	LOCAL CONST Robtarget Tr_meulage_motif_2_P33 :=[[45.7417890625,-26.569017578125,5.9224365234375],[-3.19370360057134E-06,0.00176428802739274,-0.00181018821640207,-0.999996805242986],[0,0,0,0],[8.999999E+09,8.999999E+09,8.999999E+09,8.999999E+09,8.999999E+09,8.999999E+09]];
	LOCAL CONST Robtarget Tr_meulage_motif_2_P34 :=[[46.73433984375,-26.69078125,5.9262734375],[-3.19370360057134E-06,0.00176428802739274,-0.00181018821640207,-0.999996805242986],[0,0,0,0],[8.999999E+09,8.999999E+09,8.999999E+09,8.999999E+09,8.999999E+09,8.999999E+09]];
	LOCAL CONST Robtarget Tr_meulage_motif_2_P35 :=[[47.72689453125,-26.81254296875,5.93011083984375],[-3.19370360057134E-06,0.00176428802739274,-0.00181018821640207,-0.999996805242986],[0,0,0,0],[8.999999E+09,8.999999E+09,8.999999E+09,8.999999E+09,8.999999E+09,8.999999E+09]];
	LOCAL CONST Robtarget Tr_meulage_motif_2_P36 :=[[48.72553515625,-26.823689453125,5.9303427734375],[-3.19370360057134E-06,0.00176428802739274,-0.00181018821640207,-0.999996805242986],[0,0,0,0],[8.999999E+09,8.999999E+09,8.999999E+09,8.999999E+09,8.999999E+09,8.999999E+09]];
	LOCAL CONST Robtarget Tr_meulage_motif_2_P37 :=[[49.69071484375,-26.72943359375,5.92714501953125],[-3.19370360057134E-06,0.00176428802739274,-0.00181018821640207,-0.999996805242986],[0,0,0,0],[8.999999E+09,8.999999E+09,8.999999E+09,8.999999E+09,8.999999E+09,8.999999E+09]];
	LOCAL CONST Robtarget Tr_meulage_motif_2_P38 :=[[50.57019921875,-26.563587890625,5.92162548828125],[-3.19370360057134E-06,0.00176428802739274,-0.00181018821640207,-0.999996805242986],[0,0,0,0],[8.999999E+09,8.999999E+09,8.999999E+09,8.999999E+09,8.999999E+09,8.999999E+09]];
	LOCAL CONST Robtarget Tr_meulage_motif_2_P39 :=[[51.3481640625,-26.3811640625,5.9155791015625],[-3.19370360057134E-06,0.00176428802739274,-0.00181018821640207,-0.999996805242986],[0,0,0,0],[8.999999E+09,8.999999E+09,8.999999E+09,8.999999E+09,8.999999E+09,8.999999E+09]];
	LOCAL CONST Robtarget Tr_meulage_motif_2_P40 :=[[52.5160859375,-25.904021484375,5.89987841796875],[-3.19370360057134E-06,0.00176428802739274,-0.00181018821640207,-0.999996805242986],[0,0,0,0],[8.999999E+09,8.999999E+09,8.999999E+09,8.999999E+09,8.999999E+09,8.999999E+09]];
	LOCAL CONST Robtarget Tr_meulage_motif_2_P41 :=[[53.63559765625,-25.187794921875,5.87639306640625],[-3.19370360057134E-06,0.00176428802739274,-0.00181018821640207,-0.999996805242986],[0,0,0,0],[8.999999E+09,8.999999E+09,8.999999E+09,8.999999E+09,8.999999E+09,8.999999E+09]];
	LOCAL CONST Robtarget Tr_meulage_motif_2_P42 :=[[54.601671875,-24.275298828125,5.84653271484375],[-3.19370360057134E-06,0.00176428802739274,-0.00181018821640207,-0.999996805242986],[0,0,0,0],[8.999999E+09,8.999999E+09,8.999999E+09,8.999999E+09,8.999999E+09,8.999999E+09]];
	LOCAL CONST Robtarget Tr_meulage_motif_2_P43 :=[[55.22216796875,-23.227451171875,5.8123076171875],[-3.19370360057134E-06,0.00176428802739274,-0.00181018821640207,-0.999996805242986],[0,0,0,0],[8.999999E+09,8.999999E+09,8.999999E+09,8.999999E+09,8.999999E+09,8.999999E+09]];
	LOCAL CONST Robtarget Tr_meulage_motif_2_P44 :=[[55.33381640625,-22.540328125,5.7899033203125],[-3.19370360057134E-06,0.00176428802739274,-0.00181018821640207,-0.999996805242986],[0,0,0,0],[8.999999E+09,8.999999E+09,8.999999E+09,8.999999E+09,8.999999E+09,8.999999E+09]];
	LOCAL CONST Robtarget Tr_meulage_motif_2_P45 :=[[55.41437109375,-21.8843515625,5.768517578125],[-3.19370360057134E-06,0.00176428802739274,-0.00181018821640207,-0.999996805242986],[0,0,0,0],[8.999999E+09,8.999999E+09,8.999999E+09,8.999999E+09,8.999999E+09,8.999999E+09]];
	LOCAL CONST Robtarget Tr_meulage_motif_2_P46 :=[[55.44044140625,-21.221849609375,5.7469267578125],[-3.19370360057134E-06,0.00176428802739274,-0.00181018821640207,-0.999996805242986],[0,0,0,0],[8.999999E+09,8.999999E+09,8.999999E+09,8.999999E+09,8.999999E+09,8.999999E+09]];
	LOCAL CONST Robtarget Tr_meulage_motif_2_P47 :=[[55.08015234375,-20.068220703125,5.70938330078125],[-3.19370360057134E-06,0.00176428802739274,-0.00181018821640207,-0.999996805242986],[0,0,0,0],[8.999999E+09,8.999999E+09,8.999999E+09,8.999999E+09,8.999999E+09,8.999999E+09]];
	LOCAL CONST Robtarget Tr_meulage_motif_2_P48 :=[[54.35253515625,-18.9653203125,5.673541015625],[-3.19370360057134E-06,0.00176428802739274,-0.00181018821640207,-0.999996805242986],[0,0,0,0],[8.999999E+09,8.999999E+09,8.999999E+09,8.999999E+09,8.999999E+09,8.999999E+09]];
	LOCAL CONST Robtarget Tr_meulage_motif_2_P49 :=[[53.43773046875,-18.018443359375,5.64280712890625],[-3.19370360057134E-06,0.00176428802739274,-0.00181018821640207,-0.999996805242986],[0,0,0,0],[8.999999E+09,8.999999E+09,8.999999E+09,8.999999E+09,8.999999E+09,8.999999E+09]];
	LOCAL CONST Robtarget Tr_meulage_motif_2_P50 :=[[52.80396484375,-17.542185546875,5.62737158203125],[-3.19370360057134E-06,0.00176428802739274,-0.00181018821640207,-0.999996805242986],[0,0,0,0],[8.999999E+09,8.999999E+09,8.999999E+09,8.999999E+09,8.999999E+09,8.999999E+09]];
	LOCAL CONST Robtarget Tr_meulage_motif_2_P51 :=[[51.713828125,-16.9175234375,5.60716015625],[-3.19370360057134E-06,0.00176428802739274,-0.00181018821640207,-0.999996805242986],[0,0,0,0],[8.999999E+09,8.999999E+09,8.999999E+09,8.999999E+09,8.999999E+09,8.999999E+09]];
	LOCAL CONST Robtarget Tr_meulage_motif_2_P52 :=[[50.90726171875,-16.552642578125,5.59537646484375],[-3.19370360057134E-06,0.00176428802739274,-0.00181018821640207,-0.999996805242986],[0,0,0,0],[8.999999E+09,8.999999E+09,8.999999E+09,8.999999E+09,8.999999E+09,8.999999E+09]];
	LOCAL CONST Robtarget Tr_meulage_motif_2_P53 :=[[50.00711328125,-16.2363212890625,5.5851875],[-3.19370360057134E-06,0.00176428802739274,-0.00181018821640207,-0.999996805242986],[0,0,0,0],[8.999999E+09,8.999999E+09,8.999999E+09,8.999999E+09,8.999999E+09,8.999999E+09]];
	LOCAL CONST Robtarget Tr_meulage_motif_2_P54 :=[[49.04608984375,-16.009076171875,5.5779091796875],[-3.19370360057134E-06,0.00176428802739274,-0.00181018821640207,-0.999996805242986],[0,0,0,0],[8.999999E+09,8.999999E+09,8.999999E+09,8.999999E+09,8.999999E+09,8.999999E+09]];
	LOCAL CONST Robtarget Tr_meulage_motif_2_P55 :=[[48.07439453125,-15.7785078125,5.5705234375],[-3.19370360057134E-06,0.00176428802739274,-0.00181018821640207,-0.999996805242986],[0,0,0,0],[8.999999E+09,8.999999E+09,8.999999E+09,8.999999E+09,8.999999E+09,8.999999E+09]];
	LOCAL CONST Robtarget Tr_meulage_motif_2_P56 :=[[47.08183984375,-15.6567451171875,5.56668603515625],[-3.19370360057134E-06,0.00176428802739274,-0.00181018821640207,-0.999996805242986],[0,0,0,0],[8.999999E+09,8.999999E+09,8.999999E+09,8.999999E+09,8.999999E+09,8.999999E+09]];
	LOCAL CONST Robtarget Tr_meulage_motif_2_P57 :=[[46.0892890625,-15.534982421875,5.56284912109375],[-3.19370360057134E-06,0.00176428802739274,-0.00181018821640207,-0.999996805242986],[0,0,0,0],[8.999999E+09,8.999999E+09,8.999999E+09,8.999999E+09,8.999999E+09,8.999999E+09]];
	LOCAL CONST Robtarget Tr_meulage_motif_2_P58 :=[[45.09673828125,-15.4132197265625,5.55901171875],[-3.19370360057134E-06,0.00176428802739274,-0.00181018821640207,-0.999996805242986],[0,0,0,0],[8.999999E+09,8.999999E+09,8.999999E+09,8.999999E+09,8.999999E+09,8.999999E+09]];
	LOCAL CONST Robtarget Tr_meulage_motif_2_P59 :=[[44.1041875,-15.2914580078125,5.55517431640625],[-3.19370360057134E-06,0.00176428802739274,-0.00181018821640207,-0.999996805242986],[0,0,0,0],[8.999999E+09,8.999999E+09,8.999999E+09,8.999999E+09,8.999999E+09,8.999999E+09]];
	LOCAL CONST Robtarget Tr_meulage_motif_2_P60 :=[[43.1116328125,-15.1696953125,5.5513369140625],[-3.19370360057134E-06,0.00176428802739274,-0.00181018821640207,-0.999996805242986],[0,0,0,0],[8.999999E+09,8.999999E+09,8.999999E+09,8.999999E+09,8.999999E+09,8.999999E+09]];
	LOCAL CONST Robtarget Tr_meulage_motif_2_P61 :=[[42.11908203125,-15.0479326171875,5.54749951171875],[-3.19370360057134E-06,0.00176428802739274,-0.00181018821640207,-0.999996805242986],[0,0,0,0],[8.999999E+09,8.999999E+09,8.999999E+09,8.999999E+09,8.999999E+09,8.999999E+09]];
	LOCAL CONST Robtarget Tr_meulage_motif_2_P62 :=[[41.12653125,-14.926169921875,5.54366259765625],[-3.19370360057134E-06,0.00176428802739274,-0.00181018821640207,-0.999996805242986],[0,0,0,0],[8.999999E+09,8.999999E+09,8.999999E+09,8.999999E+09,8.999999E+09,8.999999E+09]];
	LOCAL CONST Robtarget Tr_meulage_motif_2_P63 :=[[40.1339765625,-14.8044072265625,5.5398251953125],[-3.19370360057134E-06,0.00176428802739274,-0.00181018821640207,-0.999996805242986],[0,0,0,0],[8.999999E+09,8.999999E+09,8.999999E+09,8.999999E+09,8.999999E+09,8.999999E+09]];
	LOCAL CONST Robtarget Tr_meulage_motif_2_P64 :=[[39.14142578125,-14.68264453125,5.53598779296875],[-3.19370360057134E-06,0.00176428802739274,-0.00181018821640207,-0.999996805242986],[0,0,0,0],[8.999999E+09,8.999999E+09,8.999999E+09,8.999999E+09,8.999999E+09,8.999999E+09]];
	LOCAL CONST Robtarget Tr_meulage_motif_2_P65 :=[[38.148875,-14.5608828125,5.532150390625],[-3.19370360057134E-06,0.00176428802739274,-0.00181018821640207,-0.999996805242986],[0,0,0,0],[8.999999E+09,8.999999E+09,8.999999E+09,8.999999E+09,8.999999E+09,8.999999E+09]];
	LOCAL CONST Robtarget Tr_meulage_motif_2_P66 :=[[37.15632421875,-14.4391201171875,5.52831298828125],[-3.19370360057134E-06,0.00176428802739274,-0.00181018821640207,-0.999996805242986],[0,0,0,0],[8.999999E+09,8.999999E+09,8.999999E+09,8.999999E+09,8.999999E+09,8.999999E+09]];
	LOCAL CONST Robtarget Tr_meulage_motif_2_P67 :=[[36.16376953125,-14.317357421875,5.5244755859375],[-3.19370360057134E-06,0.00176428802739274,-0.00181018821640207,-0.999996805242986],[0,0,0,0],[8.999999E+09,8.999999E+09,8.999999E+09,8.999999E+09,8.999999E+09,8.999999E+09]];
	LOCAL CONST Robtarget Tr_meulage_motif_2_P68 :=[[35.17121875,-14.1955947265625,5.520638671875],[-3.19370360057134E-06,0.00176428802739274,-0.00181018821640207,-0.999996805242986],[0,0,0,0],[8.999999E+09,8.999999E+09,8.999999E+09,8.999999E+09,8.999999E+09,8.999999E+09]];
	LOCAL CONST Robtarget Tr_meulage_motif_2_P69 :=[[34.17866796875,-14.07383203125,5.51680126953125],[-3.19370360057134E-06,0.00176428802739274,-0.00181018821640207,-0.999996805242986],[0,0,0,0],[8.999999E+09,8.999999E+09,8.999999E+09,8.999999E+09,8.999999E+09,8.999999E+09]];
	LOCAL CONST Robtarget Tr_meulage_motif_2_P70 :=[[33.1861171875,-13.9520693359375,5.5129638671875],[-3.19370360057134E-06,0.00176428802739274,-0.00181018821640207,-0.999996805242986],[0,0,0,0],[8.999999E+09,8.999999E+09,8.999999E+09,8.999999E+09,8.999999E+09,8.999999E+09]];
	LOCAL CONST Robtarget Tr_meulage_motif_2_P71 :=[[32.193564453125,-13.830306640625,5.50912646484375],[-3.19370360057134E-06,0.00176428802739274,-0.00181018821640207,-0.999996805242986],[0,0,0,0],[8.999999E+09,8.999999E+09,8.999999E+09,8.999999E+09,8.999999E+09,8.999999E+09]];
	LOCAL CONST Robtarget Tr_meulage_motif_2_P72 :=[[31.20101171875,-13.708544921875,5.5052890625],[-3.19370360057134E-06,0.00176428802739274,-0.00181018821640207,-0.999996805242986],[0,0,0,0],[8.999999E+09,8.999999E+09,8.999999E+09,8.999999E+09,8.999999E+09,8.999999E+09]];
	LOCAL CONST Robtarget Tr_meulage_motif_2_P73 :=[[30.2084609375,-13.5867822265625,5.5014521484375],[-3.19370360057134E-06,0.00176428802739274,-0.00181018821640207,-0.999996805242986],[0,0,0,0],[8.999999E+09,8.999999E+09,8.999999E+09,8.999999E+09,8.999999E+09,8.999999E+09]];
	LOCAL CONST Robtarget Tr_meulage_motif_2_P74 :=[[29.215908203125,-13.46501953125,5.49761474609375],[-3.19370360057134E-06,0.00176428802739274,-0.00181018821640207,-0.999996805242986],[0,0,0,0],[8.999999E+09,8.999999E+09,8.999999E+09,8.999999E+09,8.999999E+09,8.999999E+09]];
	LOCAL CONST Robtarget Tr_meulage_motif_2_P75 :=[[28.22335546875,-13.3432568359375,5.49377734375],[-3.19370360057134E-06,0.00176428802739274,-0.00181018821640207,-0.999996805242986],[0,0,0,0],[8.999999E+09,8.999999E+09,8.999999E+09,8.999999E+09,8.999999E+09,8.999999E+09]];
	LOCAL CONST Robtarget Tr_meulage_motif_2_P76 :=[[27.2308046875,-13.221494140625,5.48993994140625],[-3.19370360057134E-06,0.00176428802739274,-0.00181018821640207,-0.999996805242986],[0,0,0,0],[8.999999E+09,8.999999E+09,8.999999E+09,8.999999E+09,8.999999E+09,8.999999E+09]];
	LOCAL CONST Robtarget Tr_meulage_motif_2_P77 :=[[26.238251953125,-13.0997314453125,5.4861025390625],[-3.19370360057134E-06,0.00176428802739274,-0.00181018821640207,-0.999996805242986],[0,0,0,0],[8.999999E+09,8.999999E+09,8.999999E+09,8.999999E+09,8.999999E+09,8.999999E+09]];
	LOCAL CONST Robtarget Tr_meulage_motif_2_P78 :=[[25.245701171875,-12.9779697265625,5.48226513671875],[-3.19370360057134E-06,0.00176428802739274,-0.00181018821640207,-0.999996805242986],[0,0,0,0],[8.999999E+09,8.999999E+09,8.999999E+09,8.999999E+09,8.999999E+09,8.999999E+09]];
	LOCAL CONST Robtarget Tr_meulage_motif_2_P79 :=[[24.2531484375,-12.85620703125,5.47842822265625],[-3.19370360057134E-06,0.00176428802739274,-0.00181018821640207,-0.999996805242986],[0,0,0,0],[8.999999E+09,8.999999E+09,8.999999E+09,8.999999E+09,8.999999E+09,8.999999E+09]];
	LOCAL CONST Robtarget Tr_meulage_motif_2_P80 :=[[23.26059765625,-12.7344443359375,5.4745908203125],[-3.19370360057134E-06,0.00176428802739274,-0.00181018821640207,-0.999996805242986],[0,0,0,0],[8.999999E+09,8.999999E+09,8.999999E+09,8.999999E+09,8.999999E+09,8.999999E+09]];
	LOCAL CONST Robtarget Tr_meulage_motif_2_P81 :=[[22.268044921875,-12.612681640625,5.47075341796875],[-3.19370360057134E-06,0.00176428802739274,-0.00181018821640207,-0.999996805242986],[0,0,0,0],[8.999999E+09,8.999999E+09,8.999999E+09,8.999999E+09,8.999999E+09,8.999999E+09]];
	LOCAL CONST Robtarget Tr_meulage_motif_2_P82 :=[[21.275494140625,-12.4909189453125,5.466916015625],[-3.19370360057134E-06,0.00176428802739274,-0.00181018821640207,-0.999996805242986],[0,0,0,0],[8.999999E+09,8.999999E+09,8.999999E+09,8.999999E+09,8.999999E+09,8.999999E+09]];
	LOCAL CONST Robtarget Tr_meulage_motif_2_P83 :=[[20.303796875,-12.2603505859375,5.45953076171875],[-3.19370360057134E-06,0.00176428802739274,-0.00181018821640207,-0.999996805242986],[0,0,0,0],[8.999999E+09,8.999999E+09,8.999999E+09,8.999999E+09,8.999999E+09,8.999999E+09]];
	LOCAL CONST Robtarget Tr_meulage_motif_2_P84 :=[[19.39007421875,-11.9355986328125,5.44906884765625],[-3.19370360057134E-06,0.00176428802739274,-0.00181018821640207,-0.999996805242986],[0,0,0,0],[8.999999E+09,8.999999E+09,8.999999E+09,8.999999E+09,8.999999E+09,8.999999E+09]];
	LOCAL CONST Robtarget Tr_meulage_motif_2_P85 :=[[18.576822265625,-11.56209375,5.4370048828125],[-3.19370360057134E-06,0.00176428802739274,-0.00181018821640207,-0.999996805242986],[0,0,0,0],[8.999999E+09,8.999999E+09,8.999999E+09,8.999999E+09,8.999999E+09,8.999999E+09]];
	LOCAL CONST Robtarget Tr_meulage_motif_2_P86 :=[[17.90767578125,-11.1737294921875,5.42443798828125],[-3.19370360057134E-06,0.00176428802739274,-0.00181018821640207,-0.999996805242986],[0,0,0,0],[8.999999E+09,8.999999E+09,8.999999E+09,8.999999E+09,8.999999E+09,8.999999E+09]];
	LOCAL CONST Robtarget Tr_meulage_motif_2_P87 :=[[16.961623046875,-10.3905224609375,5.39904150390625],[-3.19370360057134E-06,0.00176428802739274,-0.00181018821640207,-0.999996805242986],[0,0,0,0],[8.999999E+09,8.999999E+09,8.999999E+09,8.999999E+09,8.999999E+09,8.999999E+09]];
	LOCAL CONST Robtarget Tr_meulage_motif_2_P88 :=[[16.1762802734375,-9.3859560546875,5.3664111328125],[-3.19370360057134E-06,0.00176428802739274,-0.00181018821640207,-0.999996805242986],[0,0,0,0],[8.999999E+09,8.999999E+09,8.999999E+09,8.999999E+09,8.999999E+09,8.999999E+09]];
	LOCAL CONST Robtarget Tr_meulage_motif_2_P89 :=[[15.7727265625,-8.2831279296875,5.3305283203125],[-3.19370360057134E-06,0.00176428802739274,-0.00181018821640207,-0.999996805242986],[0,0,0,0],[8.999999E+09,8.999999E+09,8.999999E+09,8.999999E+09,8.999999E+09,8.999999E+09]];
	LOCAL CONST Robtarget Tr_meulage_motif_2_P90 :=[[15.673771484375,-7.57293798828125,5.30739990234375],[-3.19370360057134E-06,0.00176428802739274,-0.00181018821640207,-0.999996805242986],[0,0,0,0],[8.999999E+09,8.999999E+09,8.999999E+09,8.999999E+09,8.999999E+09,8.999999E+09]];
	LOCAL CONST Robtarget Tr_meulage_motif_2_P91 :=[[15.70420703125,-6.80130517578125,5.28225244140625],[-3.19370360057134E-06,0.00176428802739274,-0.00181018821640207,-0.999996805242986],[0,0,0,0],[8.999999E+09,8.999999E+09,8.999999E+09,8.999999E+09,8.999999E+09,8.999999E+09]];
	LOCAL CONST Robtarget Tr_meulage_motif_2_P92 :=[[15.8644345703125,-6.045720703125,5.25761083984375],[-3.19370360057134E-06,0.00176428802739274,-0.00181018821640207,-0.999996805242986],[0,0,0,0],[8.999999E+09,8.999999E+09,8.999999E+09,8.999999E+09,8.999999E+09,8.999999E+09]];
	LOCAL CONST Robtarget Tr_meulage_motif_2_P93 :=[[16.415912109375,-4.99739990234375,5.22337939453125],[-3.19370360057134E-06,0.00176428802739274,-0.00181018821640207,-0.999996805242986],[0,0,0,0],[8.999999E+09,8.999999E+09,8.999999E+09,8.999999E+09,8.999999E+09,8.999999E+09]];
	LOCAL CONST Robtarget Tr_meulage_motif_2_P94 :=[[16.898490234375,-4.4668310546875,5.20602734375],[-3.19370360057134E-06,0.00176428802739274,-0.00181018821640207,-0.999996805242986],[0,0,0,0],[8.999999E+09,8.999999E+09,8.999999E+09,8.999999E+09,8.999999E+09,8.999999E+09]];
	LOCAL CONST Robtarget Tr_meulage_motif_2_P95 :=[[17.887080078125,-3.69479956054687,5.1807412109375],[-3.19370360057134E-06,0.00176428802739274,-0.00181018821640207,-0.999996805242986],[0,0,0,0],[8.999999E+09,8.999999E+09,8.999999E+09,8.999999E+09,8.999999E+09,8.999999E+09]];
	LOCAL CONST Robtarget Tr_meulage_motif_2_P96 :=[[18.518876953125,-3.35510620117187,5.16958935546875],[-3.19370360057134E-06,0.00176428802739274,-0.00181018821640207,-0.999996805242986],[0,0,0,0],[8.999999E+09,8.999999E+09,8.999999E+09,8.999999E+09,8.999999E+09,8.999999E+09]];
	LOCAL CONST Robtarget Tr_meulage_motif_2_P97 :=[[19.694740234375,-2.951470703125,5.15628271484375],[-3.19370360057134E-06,0.00176428802739274,-0.00181018821640207,-0.999996805242986],[0,0,0,0],[8.999999E+09,8.999999E+09,8.999999E+09,8.999999E+09,8.999999E+09,8.999999E+09]];
	LOCAL CONST Robtarget Tr_meulage_motif_2_P98 :=[[20.55018359375,-2.75885375976562,5.14989404296875],[-3.19370360057134E-06,0.00176428802739274,-0.00181018821640207,-0.999996805242986],[0,0,0,0],[8.999999E+09,8.999999E+09,8.999999E+09,8.999999E+09,8.999999E+09,8.999999E+09]];
	LOCAL CONST Robtarget Tr_meulage_motif_2_P99 :=[[21.500150390625,-2.66949853515625,5.146857421875],[-3.19370360057134E-06,0.00176428802739274,-0.00181018821640207,-0.999996805242986],[0,0,0,0],[8.999999E+09,8.999999E+09,8.999999E+09,8.999999E+09,8.999999E+09,8.999999E+09]];
	LOCAL CONST Robtarget Tr_meulage_motif_2_P100 :=[[22.4876328125,-2.68128833007813,5.1471123046875],[-3.19370360057134E-06,0.00176428802739274,-0.00181018821640207,-0.999996805242986],[0,0,0,0],[8.999999E+09,8.999999E+09,8.999999E+09,8.999999E+09,8.999999E+09,8.999999E+09]];
	LOCAL CONST Robtarget Tr_meulage_motif_2_P101 :=[[23.486275390625,-2.69243359375,5.14734423828125],[-3.19370360057134E-06,0.00176428802739274,-0.00181018821640207,-0.999996805242986],[0,0,0,0],[8.999999E+09,8.999999E+09,8.999999E+09,8.999999E+09,8.999999E+09,8.999999E+09]];
	LOCAL CONST Robtarget Tr_meulage_motif_2_P102 :=[[24.478826171875,-2.81419604492188,5.151181640625],[-3.19370360057134E-06,0.00176428802739274,-0.00181018821640207,-0.999996805242986],[0,0,0,0],[8.999999E+09,8.999999E+09,8.999999E+09,8.999999E+09,8.999999E+09,8.999999E+09]];
	LOCAL CONST Robtarget Tr_meulage_motif_2_P103 :=[[25.47137890625,-2.93595849609375,5.15501904296875],[-3.19370360057134E-06,0.00176428802739274,-0.00181018821640207,-0.999996805242986],[0,0,0,0],[8.999999E+09,8.999999E+09,8.999999E+09,8.999999E+09,8.999999E+09,8.999999E+09]];
	LOCAL CONST Robtarget Tr_meulage_motif_2_P104 :=[[26.4639296875,-3.05772119140625,5.15885595703125],[-3.19370360057134E-06,0.00176428802739274,-0.00181018821640207,-0.999996805242986],[0,0,0,0],[8.999999E+09,8.999999E+09,8.999999E+09,8.999999E+09,8.999999E+09,8.999999E+09]];
	LOCAL CONST Robtarget Tr_meulage_motif_2_P105 :=[[27.456482421875,-3.17948364257813,5.162693359375],[-3.19370360057134E-06,0.00176428802739274,-0.00181018821640207,-0.999996805242986],[0,0,0,0],[8.999999E+09,8.999999E+09,8.999999E+09,8.999999E+09,8.999999E+09,8.999999E+09]];
	LOCAL CONST Robtarget Tr_meulage_motif_2_P106 :=[[28.449033203125,-3.30124609375,5.16653076171875],[-3.19370360057134E-06,0.00176428802739274,-0.00181018821640207,-0.999996805242986],[0,0,0,0],[8.999999E+09,8.999999E+09,8.999999E+09,8.999999E+09,8.999999E+09,8.999999E+09]];
	LOCAL CONST Robtarget Tr_meulage_motif_2_P107 :=[[29.4415859375,-3.4230087890625,5.1703681640625],[-3.19370360057134E-06,0.00176428802739274,-0.00181018821640207,-0.999996805242986],[0,0,0,0],[8.999999E+09,8.999999E+09,8.999999E+09,8.999999E+09,8.999999E+09,8.999999E+09]];
	LOCAL CONST Robtarget Tr_meulage_motif_2_P108 :=[[30.43413671875,-3.54477124023437,5.17420556640625],[-3.19370360057134E-06,0.00176428802739274,-0.00181018821640207,-0.999996805242986],[0,0,0,0],[8.999999E+09,8.999999E+09,8.999999E+09,8.999999E+09,8.999999E+09,8.999999E+09]];
	LOCAL CONST Robtarget Tr_meulage_motif_2_P109 :=[[31.426689453125,-3.66653393554687,5.17804296875],[-3.19370360057134E-06,0.00176428802739274,-0.00181018821640207,-0.999996805242986],[0,0,0,0],[8.999999E+09,8.999999E+09,8.999999E+09,8.999999E+09,8.999999E+09,8.999999E+09]];
	LOCAL CONST Robtarget Tr_meulage_motif_2_P110 :=[[32.419240234375,-3.78829638671875,5.1818798828125],[-3.19370360057134E-06,0.00176428802739274,-0.00181018821640207,-0.999996805242986],[0,0,0,0],[8.999999E+09,8.999999E+09,8.999999E+09,8.999999E+09,8.999999E+09,8.999999E+09]];
	LOCAL CONST Robtarget Tr_meulage_motif_2_P111 :=[[33.41179296875,-3.91005883789063,5.18571728515625],[-3.19370360057134E-06,0.00176428802739274,-0.00181018821640207,-0.999996805242986],[0,0,0,0],[8.999999E+09,8.999999E+09,8.999999E+09,8.999999E+09,8.999999E+09,8.999999E+09]];
	LOCAL CONST Robtarget Tr_meulage_motif_2_P112 :=[[34.40434375,-4.03182153320313,5.1895546875],[-3.19370360057134E-06,0.00176428802739274,-0.00181018821640207,-0.999996805242986],[0,0,0,0],[8.999999E+09,8.999999E+09,8.999999E+09,8.999999E+09,8.999999E+09,8.999999E+09]];
	LOCAL CONST Robtarget Tr_meulage_motif_2_P113 :=[[35.3968984375,-4.153583984375,5.19339208984375],[-3.19370360057134E-06,0.00176428802739274,-0.00181018821640207,-0.999996805242986],[0,0,0,0],[8.999999E+09,8.999999E+09,8.999999E+09,8.999999E+09,8.999999E+09,8.999999E+09]];
	LOCAL CONST Robtarget Tr_meulage_motif_2_P114 :=[[36.38944921875,-4.2753466796875,5.1972294921875],[-3.19370360057134E-06,0.00176428802739274,-0.00181018821640207,-0.999996805242986],[0,0,0,0],[8.999999E+09,8.999999E+09,8.999999E+09,8.999999E+09,8.999999E+09,8.999999E+09]];
	LOCAL CONST Robtarget Tr_meulage_motif_2_P115 :=[[37.382,-4.39710888671875,5.20106640625],[-3.19370360057134E-06,0.00176428802739274,-0.00181018821640207,-0.999996805242986],[0,0,0,0],[8.999999E+09,8.999999E+09,8.999999E+09,8.999999E+09,8.999999E+09,8.999999E+09]];
	LOCAL CONST Robtarget Tr_meulage_motif_2_P116 :=[[38.37455078125,-4.51887158203125,5.20490380859375],[-3.19370360057134E-06,0.00176428802739274,-0.00181018821640207,-0.999996805242986],[0,0,0,0],[8.999999E+09,8.999999E+09,8.999999E+09,8.999999E+09,8.999999E+09,8.999999E+09]];
	LOCAL CONST Robtarget Tr_meulage_motif_2_P117 :=[[39.36710546875,-4.64063427734375,5.2087412109375],[-3.19370360057134E-06,0.00176428802739274,-0.00181018821640207,-0.999996805242986],[0,0,0,0],[8.999999E+09,8.999999E+09,8.999999E+09,8.999999E+09,8.999999E+09,8.999999E+09]];
	LOCAL CONST Robtarget Tr_meulage_motif_2_P118 :=[[40.35965625,-4.762396484375,5.21257861328125],[-3.19370360057134E-06,0.00176428802739274,-0.00181018821640207,-0.999996805242986],[0,0,0,0],[8.999999E+09,8.999999E+09,8.999999E+09,8.999999E+09,8.999999E+09,8.999999E+09]];
	LOCAL CONST Robtarget Tr_meulage_motif_2_P119 :=[[41.35220703125,-4.8841591796875,5.216416015625],[-3.19370360057134E-06,0.00176428802739274,-0.00181018821640207,-0.999996805242986],[0,0,0,0],[8.999999E+09,8.999999E+09,8.999999E+09,8.999999E+09,8.999999E+09,8.999999E+09]];
	LOCAL CONST Robtarget Tr_meulage_motif_2_P120 :=[[42.3447578125,-5.005921875,5.22025341796875],[-3.19370360057134E-06,0.00176428802739274,-0.00181018821640207,-0.999996805242986],[0,0,0,0],[8.999999E+09,8.999999E+09,8.999999E+09,8.999999E+09,8.999999E+09,8.999999E+09]];
	LOCAL CONST Robtarget Tr_meulage_motif_2_P121 :=[[43.3373125,-5.1276845703125,5.22409033203125],[-3.19370360057134E-06,0.00176428802739274,-0.00181018821640207,-0.999996805242986],[0,0,0,0],[8.999999E+09,8.999999E+09,8.999999E+09,8.999999E+09,8.999999E+09,8.999999E+09]];
	LOCAL CONST Robtarget Tr_meulage_motif_2_P122 :=[[44.32986328125,-5.24944677734375,5.227927734375],[-3.19370360057134E-06,0.00176428802739274,-0.00181018821640207,-0.999996805242986],[0,0,0,0],[8.999999E+09,8.999999E+09,8.999999E+09,8.999999E+09,8.999999E+09,8.999999E+09]];
	LOCAL CONST Robtarget Tr_meulage_motif_2_P123 :=[[45.3224140625,-5.37120947265625,5.23176513671875],[-3.19370360057134E-06,0.00176428802739274,-0.00181018821640207,-0.999996805242986],[0,0,0,0],[8.999999E+09,8.999999E+09,8.999999E+09,8.999999E+09,8.999999E+09,8.999999E+09]];
	LOCAL CONST Robtarget Tr_meulage_motif_2_P124 :=[[46.31496875,-5.49297216796875,5.2356025390625],[-3.19370360057134E-06,0.00176428802739274,-0.00181018821640207,-0.999996805242986],[0,0,0,0],[8.999999E+09,8.999999E+09,8.999999E+09,8.999999E+09,8.999999E+09,8.999999E+09]];
	LOCAL CONST Robtarget Tr_meulage_motif_2_P125 :=[[47.30751953125,-5.614734375,5.23943994140625],[-3.19370360057134E-06,0.00176428802739274,-0.00181018821640207,-0.999996805242986],[0,0,0,0],[8.999999E+09,8.999999E+09,8.999999E+09,8.999999E+09,8.999999E+09,8.999999E+09]];
	LOCAL CONST Robtarget Tr_meulage_motif_2_P126 :=[[48.3000703125,-5.7364970703125,5.24327685546875],[-3.19370360057134E-06,0.00176428802739274,-0.00181018821640207,-0.999996805242986],[0,0,0,0],[8.999999E+09,8.999999E+09,8.999999E+09,8.999999E+09,8.999999E+09,8.999999E+09]];
	LOCAL CONST Robtarget Tr_meulage_motif_2_P127 :=[[49.29262109375,-5.858259765625,5.2471142578125],[-3.19370360057134E-06,0.00176428802739274,-0.00181018821640207,-0.999996805242986],[0,0,0,0],[8.999999E+09,8.999999E+09,8.999999E+09,8.999999E+09,8.999999E+09,8.999999E+09]];
	LOCAL CONST Robtarget Tr_meulage_motif_2_P128 :=[[50.28517578125,-5.98002197265625,5.25095166015625],[-3.19370360057134E-06,0.00176428802739274,-0.00181018821640207,-0.999996805242986],[0,0,0,0],[8.999999E+09,8.999999E+09,8.999999E+09,8.999999E+09,8.999999E+09,8.999999E+09]];
	LOCAL CONST Robtarget Tr_meulage_motif_2_P129 :=[[51.28381640625,-5.99116748046875,5.25118359375],[-3.19370360057134E-06,0.00176428802739274,-0.00181018821640207,-0.999996805242986],[0,0,0,0],[8.999999E+09,8.999999E+09,8.999999E+09,8.999999E+09,8.999999E+09,8.999999E+09]];
	LOCAL CONST Robtarget Tr_meulage_motif_2_P130 :=[[52.24899609375,-5.89691259765625,5.24798583984375],[-3.19370360057134E-06,0.00176428802739274,-0.00181018821640207,-0.999996805242986],[0,0,0,0],[8.999999E+09,8.999999E+09,8.999999E+09,8.999999E+09,8.999999E+09,8.999999E+09]];
	LOCAL CONST Robtarget Tr_meulage_motif_2_P131 :=[[53.12848046875,-5.73106591796875,5.24246630859375],[-3.19370360057134E-06,0.00176428802739274,-0.00181018821640207,-0.999996805242986],[0,0,0,0],[8.999999E+09,8.999999E+09,8.999999E+09,8.999999E+09,8.999999E+09,8.999999E+09]];
	LOCAL CONST Robtarget Tr_meulage_motif_2_P132 :=[[53.9064453125,-5.54864306640625,5.236419921875],[-3.19370360057134E-06,0.00176428802739274,-0.00181018821640207,-0.999996805242986],[0,0,0,0],[8.999999E+09,8.999999E+09,8.999999E+09,8.999999E+09,8.999999E+09,8.999999E+09]];
	LOCAL CONST Robtarget Tr_meulage_motif_2_P133 :=[[55.0743671875,-5.0715,5.22071923828125],[-3.19370360057134E-06,0.00176428802739274,-0.00181018821640207,-0.999996805242986],[0,0,0,0],[8.999999E+09,8.999999E+09,8.999999E+09,8.999999E+09,8.999999E+09,8.999999E+09]];
	LOCAL CONST Robtarget Tr_meulage_motif_2_P134 :=[[56.19387890625,-4.35527392578125,5.19723388671875],[-3.19370360057134E-06,0.00176428802739274,-0.00181018821640207,-0.999996805242986],[0,0,0,0],[8.999999E+09,8.999999E+09,8.999999E+09,8.999999E+09,8.999999E+09,8.999999E+09]];
	LOCAL CONST Robtarget Tr_meulage_motif_2_P135 :=[[57.159953125,-3.44277709960937,5.16737353515625],[-3.19370360057134E-06,0.00176428802739274,-0.00181018821640207,-0.999996805242986],[0,0,0,0],[8.999999E+09,8.999999E+09,8.999999E+09,8.999999E+09,8.999999E+09,8.999999E+09]];
	LOCAL CONST Robtarget Tr_meulage_motif_2_P136 :=[[57.78044921875,-2.3949306640625,5.1331484375],[-3.19370360057134E-06,0.00176428802739274,-0.00181018821640207,-0.999996805242986],[0,0,0,0],[8.999999E+09,8.999999E+09,8.999999E+09,8.999999E+09,8.999999E+09,8.999999E+09]];
	LOCAL CONST Robtarget Tr_meulage_motif_2_P137 :=[[57.89209765625,-1.70780749511719,5.110744140625],[-3.19370360057134E-06,0.00176428802739274,-0.00181018821640207,-0.999996805242986],[0,0,0,0],[8.999999E+09,8.999999E+09,8.999999E+09,8.999999E+09,8.999999E+09,8.999999E+09]];
	LOCAL CONST Robtarget Tr_meulage_motif_2_P138 :=[[57.97265234375,-1.0518310546875,5.0893583984375],[-3.19370360057134E-06,0.00176428802739274,-0.00181018821640207,-0.999996805242986],[0,0,0,0],[8.999999E+09,8.999999E+09,8.999999E+09,8.999999E+09,8.999999E+09,8.999999E+09]];
	LOCAL CONST Robtarget Tr_meulage_motif_2_P139 :=[[57.99872265625,-0.389327941894531,5.067767578125],[-3.19370360057134E-06,0.00176428802739274,-0.00181018821640207,-0.999996805242986],[0,0,0,0],[8.999999E+09,8.999999E+09,8.999999E+09,8.999999E+09,8.999999E+09,8.999999E+09]];
	LOCAL CONST Robtarget Tr_meulage_motif_2_P140 :=[[57.63843359375,0.7642998046875,5.03022412109375],[-3.19370360057134E-06,0.00176428802739274,-0.00181018821640207,-0.999996805242986],[0,0,0,0],[8.999999E+09,8.999999E+09,8.999999E+09,8.999999E+09,8.999999E+09,8.999999E+09]];
	LOCAL CONST Robtarget Tr_meulage_motif_2_P141 :=[[56.91081640625,1.86720166015625,4.9943818359375],[-3.19370360057134E-06,0.00176428802739274,-0.00181018821640207,-0.999996805242986],[0,0,0,0],[8.999999E+09,8.999999E+09,8.999999E+09,8.999999E+09,8.999999E+09,8.999999E+09]];
	LOCAL CONST Robtarget Tr_meulage_motif_2_P142 :=[[55.99601171875,2.81407861328125,4.96364794921875],[-3.19370360057134E-06,0.00176428802739274,-0.00181018821640207,-0.999996805242986],[0,0,0,0],[8.999999E+09,8.999999E+09,8.999999E+09,8.999999E+09,8.999999E+09,8.999999E+09]];
	LOCAL CONST Robtarget Tr_meulage_motif_2_P143 :=[[55.36224609375,3.29033471679688,4.94821240234375],[-3.19370360057134E-06,0.00176428802739274,-0.00181018821640207,-0.999996805242986],[0,0,0,0],[8.999999E+09,8.999999E+09,8.999999E+09,8.999999E+09,8.999999E+09,8.999999E+09]];
	LOCAL CONST Robtarget Tr_meulage_motif_2_P144 :=[[54.272109375,3.914998046875,4.9280009765625],[-3.19370360057134E-06,0.00176428802739274,-0.00181018821640207,-0.999996805242986],[0,0,0,0],[8.999999E+09,8.999999E+09,8.999999E+09,8.999999E+09,8.999999E+09,8.999999E+09]];
	LOCAL CONST Robtarget Tr_meulage_motif_2_P145 :=[[53.46554296875,4.27987890625,4.91621728515625],[-3.19370360057134E-06,0.00176428802739274,-0.00181018821640207,-0.999996805242986],[0,0,0,0],[8.999999E+09,8.999999E+09,8.999999E+09,8.999999E+09,8.999999E+09,8.999999E+09]];
	LOCAL CONST Robtarget Tr_meulage_motif_2_P146 :=[[52.56539453125,4.59619921875,4.9060283203125],[-3.19370360057134E-06,0.00176428802739274,-0.00181018821640207,-0.999996805242986],[0,0,0,0],[8.999999E+09,8.999999E+09,8.999999E+09,8.999999E+09,8.999999E+09,8.999999E+09]];
	LOCAL CONST Robtarget Tr_meulage_motif_2_P147 :=[[51.60437109375,4.82344482421875,4.89875],[-3.19370360057134E-06,0.00176428802739274,-0.00181018821640207,-0.999996805242986],[0,0,0,0],[8.999999E+09,8.999999E+09,8.999999E+09,8.999999E+09,8.999999E+09,8.999999E+09]];
	LOCAL CONST Robtarget Tr_meulage_motif_2_P148 :=[[50.63267578125,5.05401318359375,4.8913642578125],[-3.19370360057134E-06,0.00176428802739274,-0.00181018821640207,-0.999996805242986],[0,0,0,0],[8.999999E+09,8.999999E+09,8.999999E+09,8.999999E+09,8.999999E+09,8.999999E+09]];
	LOCAL CONST Robtarget Tr_meulage_motif_2_P149 :=[[49.64012109375,5.17577587890625,4.88752685546875],[-3.19370360057134E-06,0.00176428802739274,-0.00181018821640207,-0.999996805242986],[0,0,0,0],[8.999999E+09,8.999999E+09,8.999999E+09,8.999999E+09,8.999999E+09,8.999999E+09]];
	LOCAL CONST Robtarget Tr_meulage_motif_2_P150 :=[[48.6475703125,5.29753857421875,4.88368994140625],[-3.19370360057134E-06,0.00176428802739274,-0.00181018821640207,-0.999996805242986],[0,0,0,0],[8.999999E+09,8.999999E+09,8.999999E+09,8.999999E+09,8.999999E+09,8.999999E+09]];
	LOCAL CONST Robtarget Tr_meulage_motif_2_P151 :=[[47.65501953125,5.41930078125,4.8798525390625],[-3.19370360057134E-06,0.00176428802739274,-0.00181018821640207,-0.999996805242986],[0,0,0,0],[8.999999E+09,8.999999E+09,8.999999E+09,8.999999E+09,8.999999E+09,8.999999E+09]];
	LOCAL CONST Robtarget Tr_meulage_motif_2_P152 :=[[46.66246875,5.5410634765625,4.87601513671875],[-3.19370360057134E-06,0.00176428802739274,-0.00181018821640207,-0.999996805242986],[0,0,0,0],[8.999999E+09,8.999999E+09,8.999999E+09,8.999999E+09,8.999999E+09,8.999999E+09]];
	LOCAL CONST Robtarget Tr_meulage_motif_2_P153 :=[[45.6699140625,5.662826171875,4.872177734375],[-3.19370360057134E-06,0.00176428802739274,-0.00181018821640207,-0.999996805242986],[0,0,0,0],[8.999999E+09,8.999999E+09,8.999999E+09,8.999999E+09,8.999999E+09,8.999999E+09]];
	LOCAL CONST Robtarget Tr_meulage_motif_2_P154 :=[[44.67736328125,5.7845888671875,4.86834033203125],[-3.19370360057134E-06,0.00176428802739274,-0.00181018821640207,-0.999996805242986],[0,0,0,0],[8.999999E+09,8.999999E+09,8.999999E+09,8.999999E+09,8.999999E+09,8.999999E+09]];
	LOCAL CONST Robtarget Tr_meulage_motif_2_P155 :=[[43.6848125,5.90635107421875,4.8645029296875],[-3.19370360057134E-06,0.00176428802739274,-0.00181018821640207,-0.999996805242986],[0,0,0,0],[8.999999E+09,8.999999E+09,8.999999E+09,8.999999E+09,8.999999E+09,8.999999E+09]];
	LOCAL CONST Robtarget Tr_meulage_motif_2_P156 :=[[42.69226171875,6.02811376953125,4.860666015625],[-3.19370360057134E-06,0.00176428802739274,-0.00181018821640207,-0.999996805242986],[0,0,0,0],[8.999999E+09,8.999999E+09,8.999999E+09,8.999999E+09,8.999999E+09,8.999999E+09]];
	LOCAL CONST Robtarget Tr_meulage_motif_2_P157 :=[[41.69970703125,6.14987646484375,4.85682861328125],[-3.19370360057134E-06,0.00176428802739274,-0.00181018821640207,-0.999996805242986],[0,0,0,0],[8.999999E+09,8.999999E+09,8.999999E+09,8.999999E+09,8.999999E+09,8.999999E+09]];
	LOCAL CONST Robtarget Tr_meulage_motif_2_P158 :=[[40.70715625,6.271638671875,4.8529912109375],[-3.19370360057134E-06,0.00176428802739274,-0.00181018821640207,-0.999996805242986],[0,0,0,0],[8.999999E+09,8.999999E+09,8.999999E+09,8.999999E+09,8.999999E+09,8.999999E+09]];
	LOCAL CONST Robtarget Tr_meulage_motif_2_P159 :=[[39.71460546875,6.3934013671875,4.84915380859375],[-3.19370360057134E-06,0.00176428802739274,-0.00181018821640207,-0.999996805242986],[0,0,0,0],[8.999999E+09,8.999999E+09,8.999999E+09,8.999999E+09,8.999999E+09,8.999999E+09]];
	LOCAL CONST Robtarget Tr_meulage_motif_2_P160 :=[[38.72205078125,6.5151640625,4.84531640625],[-3.19370360057134E-06,0.00176428802739274,-0.00181018821640207,-0.999996805242986],[0,0,0,0],[8.999999E+09,8.999999E+09,8.999999E+09,8.999999E+09,8.999999E+09,8.999999E+09]];
	LOCAL CONST Robtarget Tr_meulage_motif_2_P161 :=[[37.7295,6.63692626953125,4.8414794921875],[-3.19370360057134E-06,0.00176428802739274,-0.00181018821640207,-0.999996805242986],[0,0,0,0],[8.999999E+09,8.999999E+09,8.999999E+09,8.999999E+09,8.999999E+09,8.999999E+09]];
	LOCAL CONST Robtarget Tr_meulage_motif_2_P162 :=[[36.73694921875,6.75868896484375,4.83764208984375],[-3.19370360057134E-06,0.00176428802739274,-0.00181018821640207,-0.999996805242986],[0,0,0,0],[8.999999E+09,8.999999E+09,8.999999E+09,8.999999E+09,8.999999E+09,8.999999E+09]];
	LOCAL CONST Robtarget Tr_meulage_motif_2_P163 :=[[35.7443984375,6.88045166015625,4.8338046875],[-3.19370360057134E-06,0.00176428802739274,-0.00181018821640207,-0.999996805242986],[0,0,0,0],[8.999999E+09,8.999999E+09,8.999999E+09,8.999999E+09,8.999999E+09,8.999999E+09]];
	LOCAL CONST Robtarget Tr_meulage_motif_2_P164 :=[[34.75184375,7.0022138671875,4.82996728515625],[-3.19370360057134E-06,0.00176428802739274,-0.00181018821640207,-0.999996805242986],[0,0,0,0],[8.999999E+09,8.999999E+09,8.999999E+09,8.999999E+09,8.999999E+09,8.999999E+09]];
	LOCAL CONST Robtarget Tr_meulage_motif_2_P165 :=[[33.75929296875,7.1239765625,4.8261298828125],[-3.19370360057134E-06,0.00176428802739274,-0.00181018821640207,-0.999996805242986],[0,0,0,0],[8.999999E+09,8.999999E+09,8.999999E+09,8.999999E+09,8.999999E+09,8.999999E+09]];
	LOCAL CONST Robtarget Tr_meulage_motif_2_P166 :=[[32.7667421875,7.2457392578125,4.82229248046875],[-3.19370360057134E-06,0.00176428802739274,-0.00181018821640207,-0.999996805242986],[0,0,0,0],[8.999999E+09,8.999999E+09,8.999999E+09,8.999999E+09,8.999999E+09,8.999999E+09]];
	LOCAL CONST Robtarget Tr_meulage_motif_2_P167 :=[[31.774189453125,7.367501953125,4.81845556640625],[-3.19370360057134E-06,0.00176428802739274,-0.00181018821640207,-0.999996805242986],[0,0,0,0],[8.999999E+09,8.999999E+09,8.999999E+09,8.999999E+09,8.999999E+09,8.999999E+09]];
	LOCAL CONST Robtarget Tr_meulage_motif_2_P168 :=[[30.781638671875,7.48926416015625,4.8146181640625],[-3.19370360057134E-06,0.00176428802739274,-0.00181018821640207,-0.999996805242986],[0,0,0,0],[8.999999E+09,8.999999E+09,8.999999E+09,8.999999E+09,8.999999E+09,8.999999E+09]];
	LOCAL CONST Robtarget Tr_meulage_motif_2_P169 :=[[29.7890859375,7.61102685546875,4.81078076171875],[-3.19370360057134E-06,0.00176428802739274,-0.00181018821640207,-0.999996805242986],[0,0,0,0],[8.999999E+09,8.999999E+09,8.999999E+09,8.999999E+09,8.999999E+09,8.999999E+09]];
	LOCAL CONST Robtarget Tr_meulage_motif_2_P170 :=[[28.796533203125,7.73278955078125,4.806943359375],[-3.19370360057134E-06,0.00176428802739274,-0.00181018821640207,-0.999996805242986],[0,0,0,0],[8.999999E+09,8.999999E+09,8.999999E+09,8.999999E+09,8.999999E+09,8.999999E+09]];
	LOCAL CONST Robtarget Tr_meulage_motif_2_P171 :=[[27.803982421875,7.8545517578125,4.80310595703125],[-3.19370360057134E-06,0.00176428802739274,-0.00181018821640207,-0.999996805242986],[0,0,0,0],[8.999999E+09,8.999999E+09,8.999999E+09,8.999999E+09,8.999999E+09,8.999999E+09]];
	LOCAL CONST Robtarget Tr_meulage_motif_2_P172 :=[[26.8114296875,7.976314453125,4.79926904296875],[-3.19370360057134E-06,0.00176428802739274,-0.00181018821640207,-0.999996805242986],[0,0,0,0],[8.999999E+09,8.999999E+09,8.999999E+09,8.999999E+09,8.999999E+09,8.999999E+09]];
	LOCAL CONST Robtarget Tr_meulage_motif_2_P173 :=[[25.81887890625,8.0980771484375,4.795431640625],[-3.19370360057134E-06,0.00176428802739274,-0.00181018821640207,-0.999996805242986],[0,0,0,0],[8.999999E+09,8.999999E+09,8.999999E+09,8.999999E+09,8.999999E+09,8.999999E+09]];
	LOCAL CONST Robtarget Tr_meulage_motif_2_P174 :=[[24.826326171875,8.21983984375,4.79159423828125],[-3.19370360057134E-06,0.00176428802739274,-0.00181018821640207,-0.999996805242986],[0,0,0,0],[8.999999E+09,8.999999E+09,8.999999E+09,8.999999E+09,8.999999E+09,8.999999E+09]];
	LOCAL CONST Robtarget Tr_meulage_motif_2_P175 :=[[23.833775390625,8.3416025390625,4.7877568359375],[-3.19370360057134E-06,0.00176428802739274,-0.00181018821640207,-0.999996805242986],[0,0,0,0],[8.999999E+09,8.999999E+09,8.999999E+09,8.999999E+09,8.999999E+09,8.999999E+09]];
	LOCAL CONST Robtarget Tr_meulage_motif_2_P176 :=[[22.862078125,8.5721708984375,4.78037158203125],[-3.19370360057134E-06,0.00176428802739274,-0.00181018821640207,-0.999996805242986],[0,0,0,0],[8.999999E+09,8.999999E+09,8.999999E+09,8.999999E+09,8.999999E+09,8.999999E+09]];
	LOCAL CONST Robtarget Tr_meulage_motif_2_P177 :=[[21.94835546875,8.896921875,4.7699091796875],[-3.19370360057134E-06,0.00176428802739274,-0.00181018821640207,-0.999996805242986],[0,0,0,0],[8.999999E+09,8.999999E+09,8.999999E+09,8.999999E+09,8.999999E+09,8.999999E+09]];
	LOCAL CONST Robtarget Tr_meulage_motif_2_P178 :=[[21.135103515625,9.2704267578125,4.757845703125],[-3.19370360057134E-06,0.00176428802739274,-0.00181018821640207,-0.999996805242986],[0,0,0,0],[8.999999E+09,8.999999E+09,8.999999E+09,8.999999E+09,8.999999E+09,8.999999E+09]];
	LOCAL CONST Robtarget Tr_meulage_motif_2_P179 :=[[20.465955078125,9.6587763671875,4.745279296875],[-3.19370360057134E-06,0.00176428802739274,-0.00181018821640207,-0.999996805242986],[0,0,0,0],[8.999999E+09,8.999999E+09,8.999999E+09,8.999999E+09,8.999999E+09,8.999999E+09]];
	LOCAL CONST Robtarget Tr_meulage_motif_2_P180 :=[[19.51990234375,10.4419833984375,4.7198828125],[-3.19370360057134E-06,0.00176428802739274,-0.00181018821640207,-0.999996805242986],[0,0,0,0],[8.999999E+09,8.999999E+09,8.999999E+09,8.999999E+09,8.999999E+09,8.999999E+09]];
	LOCAL CONST Robtarget Tr_meulage_motif_2_P181 :=[[18.734560546875,11.4465654296875,4.68725146484375],[-3.19370360057134E-06,0.00176428802739274,-0.00181018821640207,-0.999996805242986],[0,0,0,0],[8.999999E+09,8.999999E+09,8.999999E+09,8.999999E+09,8.999999E+09,8.999999E+09]];
	LOCAL CONST Robtarget Tr_meulage_motif_2_P182 :=[[18.331005859375,12.5493779296875,4.65136962890625],[-3.19370360057134E-06,0.00176428802739274,-0.00181018821640207,-0.999996805242986],[0,0,0,0],[8.999999E+09,8.999999E+09,8.999999E+09,8.999999E+09,8.999999E+09,8.999999E+09]];
	LOCAL CONST Robtarget Tr_meulage_motif_2_P183 :=[[18.232052734375,13.2595830078125,4.62824072265625],[-3.19370360057134E-06,0.00176428802739274,-0.00181018821640207,-0.999996805242986],[0,0,0,0],[8.999999E+09,8.999999E+09,8.999999E+09,8.999999E+09,8.999999E+09,8.999999E+09]];
	LOCAL CONST Robtarget Tr_meulage_motif_2_P184 :=[[18.26248828125,14.0312158203125,4.60309326171875],[-3.19370360057134E-06,0.00176428802739274,-0.00181018821640207,-0.999996805242986],[0,0,0,0],[8.999999E+09,8.999999E+09,8.999999E+09,8.999999E+09,8.999999E+09,8.999999E+09]];
	LOCAL CONST Robtarget Tr_meulage_motif_2_P185 :=[[18.422712890625,14.78678515625,4.5784521484375],[-3.19370360057134E-06,0.00176428802739274,-0.00181018821640207,-0.999996805242986],[0,0,0,0],[8.999999E+09,8.999999E+09,8.999999E+09,8.999999E+09,8.999999E+09,8.999999E+09]];
	LOCAL CONST Robtarget Tr_meulage_motif_2_P186 :=[[18.974193359375,15.83510546875,4.544220703125],[-3.19370360057134E-06,0.00176428802739274,-0.00181018821640207,-0.999996805242986],[0,0,0,0],[8.999999E+09,8.999999E+09,8.999999E+09,8.999999E+09,8.999999E+09,8.999999E+09]];
	LOCAL CONST Robtarget Tr_meulage_motif_2_P187 :=[[19.45676953125,16.3656748046875,4.52686865234375],[-3.19370360057134E-06,0.00176428802739274,-0.00181018821640207,-0.999996805242986],[0,0,0,0],[8.999999E+09,8.999999E+09,8.999999E+09,8.999999E+09,8.999999E+09,8.999999E+09]];
	LOCAL CONST Robtarget Tr_meulage_motif_2_P188 :=[[20.44536328125,17.137736328125,4.50158154296875],[-3.19370360057134E-06,0.00176428802739274,-0.00181018821640207,-0.999996805242986],[0,0,0,0],[8.999999E+09,8.999999E+09,8.999999E+09,8.999999E+09,8.999999E+09,8.999999E+09]];
	LOCAL CONST Robtarget Tr_meulage_motif_2_P189 :=[[21.07715625,17.477400390625,4.4904306640625],[-3.19370360057134E-06,0.00176428802739274,-0.00181018821640207,-0.999996805242986],[0,0,0,0],[8.999999E+09,8.999999E+09,8.999999E+09,8.999999E+09,8.999999E+09,8.999999E+09]];
	LOCAL CONST Robtarget Tr_meulage_motif_2_P190 :=[[22.2530234375,17.88106640625,4.477123046875],[-3.19370360057134E-06,0.00176428802739274,-0.00181018821640207,-0.999996805242986],[0,0,0,0],[8.999999E+09,8.999999E+09,8.999999E+09,8.999999E+09,8.999999E+09,8.999999E+09]];
	LOCAL CONST Robtarget Tr_meulage_motif_2_P191 :=[[23.108466796875,18.07368359375,4.470734375],[-3.19370360057134E-06,0.00176428802739274,-0.00181018821640207,-0.999996805242986],[0,0,0,0],[8.999999E+09,8.999999E+09,8.999999E+09,8.999999E+09,8.999999E+09,8.999999E+09]];
	LOCAL CONST Robtarget Tr_meulage_motif_2_P192 :=[[24.058435546875,18.1630546875,4.467697265625],[-3.19370360057134E-06,0.00176428802739274,-0.00181018821640207,-0.999996805242986],[0,0,0,0],[8.999999E+09,8.999999E+09,8.999999E+09,8.999999E+09,8.999999E+09,8.999999E+09]];
	LOCAL CONST Robtarget Tr_meulage_motif_2_P193 :=[[25.045912109375,18.151216796875,4.46795361328125],[-3.19370360057134E-06,0.00176428802739274,-0.00181018821640207,-0.999996805242986],[0,0,0,0],[8.999999E+09,8.999999E+09,8.999999E+09,8.999999E+09,8.999999E+09,8.999999E+09]];
	LOCAL CONST Robtarget Tr_meulage_motif_2_P194 :=[[26.044556640625,18.140087890625,4.46818505859375],[-3.19370360057134E-06,0.00176428802739274,-0.00181018821640207,-0.999996805242986],[0,0,0,0],[8.999999E+09,8.999999E+09,8.999999E+09,8.999999E+09,8.999999E+09,8.999999E+09]];
	LOCAL CONST Robtarget Tr_meulage_motif_2_P195 :=[[27.037107421875,18.01832421875,4.4720224609375],[-3.19370360057134E-06,0.00176428802739274,-0.00181018821640207,-0.999996805242986],[0,0,0,0],[8.999999E+09,8.999999E+09,8.999999E+09,8.999999E+09,8.999999E+09,8.999999E+09]];
	LOCAL CONST Robtarget Tr_meulage_motif_2_P196 :=[[28.02966015625,17.8965625,4.47585986328125],[-3.19370360057134E-06,0.00176428802739274,-0.00181018821640207,-0.999996805242986],[0,0,0,0],[8.999999E+09,8.999999E+09,8.999999E+09,8.999999E+09,8.999999E+09,8.999999E+09]];
	LOCAL CONST Robtarget Tr_meulage_motif_2_P197 :=[[29.0222109375,17.77480078125,4.47969677734375],[-3.19370360057134E-06,0.00176428802739274,-0.00181018821640207,-0.999996805242986],[0,0,0,0],[8.999999E+09,8.999999E+09,8.999999E+09,8.999999E+09,8.999999E+09,8.999999E+09]];
	LOCAL CONST Robtarget Tr_meulage_motif_2_P198 :=[[30.014763671875,17.653037109375,4.4835341796875],[-3.19370360057134E-06,0.00176428802739274,-0.00181018821640207,-0.999996805242986],[0,0,0,0],[8.999999E+09,8.999999E+09,8.999999E+09,8.999999E+09,8.999999E+09,8.999999E+09]];
	LOCAL CONST Robtarget Tr_meulage_motif_2_P199 :=[[31.007314453125,17.531275390625,4.48737158203125],[-3.19370360057134E-06,0.00176428802739274,-0.00181018821640207,-0.999996805242986],[0,0,0,0],[8.999999E+09,8.999999E+09,8.999999E+09,8.999999E+09,8.999999E+09,8.999999E+09]];
	LOCAL CONST Robtarget Tr_meulage_motif_2_P200 :=[[31.9998671875,17.40951171875,4.491208984375],[-3.19370360057134E-06,0.00176428802739274,-0.00181018821640207,-0.999996805242986],[0,0,0,0],[8.999999E+09,8.999999E+09,8.999999E+09,8.999999E+09,8.999999E+09,8.999999E+09]];
	LOCAL CONST Robtarget Tr_meulage_motif_2_P201 :=[[32.99241796875,17.28775,4.49504638671875],[-3.19370360057134E-06,0.00176428802739274,-0.00181018821640207,-0.999996805242986],[0,0,0,0],[8.999999E+09,8.999999E+09,8.999999E+09,8.999999E+09,8.999999E+09,8.999999E+09]];
	LOCAL CONST Robtarget Tr_meulage_motif_2_P202 :=[[33.98496875,17.16598828125,4.49888330078125],[-3.19370360057134E-06,0.00176428802739274,-0.00181018821640207,-0.999996805242986],[0,0,0,0],[8.999999E+09,8.999999E+09,8.999999E+09,8.999999E+09,8.999999E+09,8.999999E+09]];
	LOCAL CONST Robtarget Tr_meulage_motif_2_P203 :=[[34.9775234375,17.044224609375,4.502720703125],[-3.19370360057134E-06,0.00176428802739274,-0.00181018821640207,-0.999996805242986],[0,0,0,0],[8.999999E+09,8.999999E+09,8.999999E+09,8.999999E+09,8.999999E+09,8.999999E+09]];
	LOCAL CONST Robtarget Tr_meulage_motif_2_P204 :=[[35.97007421875,16.922462890625,4.50655810546875],[-3.19370360057134E-06,0.00176428802739274,-0.00181018821640207,-0.999996805242986],[0,0,0,0],[8.999999E+09,8.999999E+09,8.999999E+09,8.999999E+09,8.999999E+09,8.999999E+09]];
	LOCAL CONST Robtarget Tr_meulage_motif_2_P205 :=[[36.962625,16.80069921875,4.5103955078125],[-3.19370360057134E-06,0.00176428802739274,-0.00181018821640207,-0.999996805242986],[0,0,0,0],[8.999999E+09,8.999999E+09,8.999999E+09,8.999999E+09,8.999999E+09,8.999999E+09]];
	LOCAL CONST Robtarget Tr_meulage_motif_2_P206 :=[[37.9551796875,16.6789375,4.51423291015625],[-3.19370360057134E-06,0.00176428802739274,-0.00181018821640207,-0.999996805242986],[0,0,0,0],[8.999999E+09,8.999999E+09,8.999999E+09,8.999999E+09,8.999999E+09,8.999999E+09]];
	LOCAL CONST Robtarget Tr_meulage_motif_2_P207 :=[[38.94773046875,16.557173828125,4.5180703125],[-3.19370360057134E-06,0.00176428802739274,-0.00181018821640207,-0.999996805242986],[0,0,0,0],[8.999999E+09,8.999999E+09,8.999999E+09,8.999999E+09,8.999999E+09,8.999999E+09]];
	LOCAL CONST Robtarget Tr_meulage_motif_2_P208 :=[[39.94028125,16.435412109375,4.5219072265625],[-3.19370360057134E-06,0.00176428802739274,-0.00181018821640207,-0.999996805242986],[0,0,0,0],[8.999999E+09,8.999999E+09,8.999999E+09,8.999999E+09,8.999999E+09,8.999999E+09]];
	LOCAL CONST Robtarget Tr_meulage_motif_2_P209 :=[[40.93283203125,16.3136494140625,4.52574462890625],[-3.19370360057134E-06,0.00176428802739274,-0.00181018821640207,-0.999996805242986],[0,0,0,0],[8.999999E+09,8.999999E+09,8.999999E+09,8.999999E+09,8.999999E+09,8.999999E+09]];
	LOCAL CONST Robtarget Tr_meulage_motif_2_P210 :=[[41.92538671875,16.19188671875,4.52958203125],[-3.19370360057134E-06,0.00176428802739274,-0.00181018821640207,-0.999996805242986],[0,0,0,0],[8.999999E+09,8.999999E+09,8.999999E+09,8.999999E+09,8.999999E+09,8.999999E+09]];
	LOCAL CONST Robtarget Tr_meulage_motif_2_P211 :=[[42.9179375,16.0701240234375,4.53341943359375],[-3.19370360057134E-06,0.00176428802739274,-0.00181018821640207,-0.999996805242986],[0,0,0,0],[8.999999E+09,8.999999E+09,8.999999E+09,8.999999E+09,8.999999E+09,8.999999E+09]];
	LOCAL CONST Robtarget Tr_meulage_motif_2_P212 :=[[43.91048828125,15.9483623046875,4.5372568359375],[-3.19370360057134E-06,0.00176428802739274,-0.00181018821640207,-0.999996805242986],[0,0,0,0],[8.999999E+09,8.999999E+09,8.999999E+09,8.999999E+09,8.999999E+09,8.999999E+09]];
	LOCAL CONST Robtarget Tr_meulage_motif_2_P213 :=[[44.9030390625,15.826599609375,4.54109375],[-3.19370360057134E-06,0.00176428802739274,-0.00181018821640207,-0.999996805242986],[0,0,0,0],[8.999999E+09,8.999999E+09,8.999999E+09,8.999999E+09,8.999999E+09,8.999999E+09]];
	LOCAL CONST Robtarget Tr_meulage_motif_2_P214 :=[[45.89559375,15.7048369140625,4.54493115234375],[-3.19370360057134E-06,0.00176428802739274,-0.00181018821640207,-0.999996805242986],[0,0,0,0],[8.999999E+09,8.999999E+09,8.999999E+09,8.999999E+09,8.999999E+09,8.999999E+09]];
	LOCAL CONST Robtarget Tr_meulage_motif_2_P215 :=[[46.88814453125,15.58307421875,4.5487685546875],[-3.19370360057134E-06,0.00176428802739274,-0.00181018821640207,-0.999996805242986],[0,0,0,0],[8.999999E+09,8.999999E+09,8.999999E+09,8.999999E+09,8.999999E+09,8.999999E+09]];
	LOCAL CONST Robtarget Tr_meulage_motif_2_P216 :=[[47.8806953125,15.4613115234375,4.55260595703125],[-3.19370360057134E-06,0.00176428802739274,-0.00181018821640207,-0.999996805242986],[0,0,0,0],[8.999999E+09,8.999999E+09,8.999999E+09,8.999999E+09,8.999999E+09,8.999999E+09]];
	LOCAL CONST Robtarget Tr_meulage_motif_2_P217 :=[[48.87325,15.339548828125,4.556443359375],[-3.19370360057134E-06,0.00176428802739274,-0.00181018821640207,-0.999996805242986],[0,0,0,0],[8.999999E+09,8.999999E+09,8.999999E+09,8.999999E+09,8.999999E+09,8.999999E+09]];
	LOCAL CONST Robtarget Tr_meulage_motif_2_P218 :=[[49.86580078125,15.217787109375,4.56028076171875],[-3.19370360057134E-06,0.00176428802739274,-0.00181018821640207,-0.999996805242986],[0,0,0,0],[8.999999E+09,8.999999E+09,8.999999E+09,8.999999E+09,8.999999E+09,8.999999E+09]];
	LOCAL CONST Robtarget Tr_meulage_motif_2_P219 :=[[50.8583515625,15.0960244140625,4.56411767578125],[-3.19370360057134E-06,0.00176428802739274,-0.00181018821640207,-0.999996805242986],[0,0,0,0],[8.999999E+09,8.999999E+09,8.999999E+09,8.999999E+09,8.999999E+09,8.999999E+09]];
	LOCAL CONST Robtarget Tr_meulage_motif_2_P220 :=[[51.85090234375,14.97426171875,4.567955078125],[-3.19370360057134E-06,0.00176428802739274,-0.00181018821640207,-0.999996805242986],[0,0,0,0],[8.999999E+09,8.999999E+09,8.999999E+09,8.999999E+09,8.999999E+09,8.999999E+09]];
	LOCAL CONST Robtarget Tr_meulage_motif_2_P221 :=[[52.84345703125,14.8524990234375,4.57179248046875],[-3.19370360057134E-06,0.00176428802739274,-0.00181018821640207,-0.999996805242986],[0,0,0,0],[8.999999E+09,8.999999E+09,8.999999E+09,8.999999E+09,8.999999E+09,8.999999E+09]];
	LOCAL CONST Robtarget Tr_meulage_motif_2_P222 :=[[53.8360078125,14.730736328125,4.5756298828125],[-3.19370360057134E-06,0.00176428802739274,-0.00181018821640207,-0.999996805242986],[0,0,0,0],[8.999999E+09,8.999999E+09,8.999999E+09,8.999999E+09,8.999999E+09,8.999999E+09]];
	LOCAL CONST Robtarget Tr_meulage_motif_2_P223 :=[[54.82855859375,14.6089736328125,4.57946728515625],[-3.19370360057134E-06,0.00176428802739274,-0.00181018821640207,-0.999996805242986],[0,0,0,0],[8.999999E+09,8.999999E+09,8.999999E+09,8.999999E+09,8.999999E+09,8.999999E+09]];
	LOCAL CONST Robtarget Tr_meulage_motif_2_P224 :=[[55.827203125,14.5978447265625,4.57969873046875],[-3.19370360057134E-06,0.00176428802739274,-0.00181018821640207,-0.999996805242986],[0,0,0,0],[8.999999E+09,8.999999E+09,8.999999E+09,8.999999E+09,8.999999E+09,8.999999E+09]];
	LOCAL CONST Robtarget Tr_meulage_motif_2_P225 :=[[56.8146796875,14.5860078125,4.57995458984375],[-3.19370360057134E-06,0.00176428802739274,-0.00181018821640207,-0.999996805242986],[0,0,0,0],[8.999999E+09,8.999999E+09,8.999999E+09,8.999999E+09,8.999999E+09,8.999999E+09]];
	LOCAL CONST Robtarget Tr_meulage_motif_2_P226 :=[[57.79922265625,14.5626201171875,4.58058740234375],[-3.19370360057134E-06,0.00176428802739274,-0.00181018821640207,-0.999996805242986],[0,0,0,0],[8.999999E+09,8.999999E+09,8.999999E+09,8.999999E+09,8.999999E+09,8.999999E+09]];
	LOCAL CONST Robtarget Tr_meulage_motif_2_P227 :=[[58.77215234375,14.581015625,4.5798603515625],[-3.19370360057134E-06,0.00176428802739274,-0.00181018821640207,-0.999996805242986],[0,0,0,0],[8.999999E+09,8.999999E+09,8.999999E+09,8.999999E+09,8.999999E+09,8.999999E+09]];
	LOCAL CONST Robtarget Tr_meulage_motif_2_P228 :=[[59.946171875,14.68659375,4.57626611328125],[-3.19370360057134E-06,0.00176428802739274,-0.00181018821640207,-0.999996805242986],[0,0,0,0],[8.999999E+09,8.999999E+09,8.999999E+09,8.999999E+09,8.999999E+09,8.999999E+09]];
	LOCAL CONST Robtarget Tr_meulage_motif_2_P229 :=[[60.90286328125,14.88634765625,4.56963134765625],[-3.19370360057134E-06,0.00176428802739274,-0.00181018821640207,-0.999996805242986],[0,0,0,0],[8.999999E+09,8.999999E+09,8.999999E+09,8.999999E+09,8.999999E+09,8.999999E+09]];
	LOCAL CONST Robtarget Tr_meulage_motif_2_degg1 :=[[60.9381488134443,14.8501438948919,-5.4302408624713],[-3.19370360057134E-06,0.00176428802739274,-0.00181018821640207,-0.999996805242986],[0,0,0,0],[8.999999E+09,8.999999E+09,8.999999E+09,8.999999E+09,8.999999E+09,8.999999E+09]];
	LOCAL CONST Robtarget Tr_meulage_motif_2_degg2 :=[[61.6085739251366,14.1622724290886,-195.427812854895],[-3.19370360057134E-06,0.00176428802739274,-0.00181018821640207,-0.999996805242986],[0,0,0,0],[8.999999E+09,8.999999E+09,8.999999E+09,8.999999E+09,8.999999E+09,8.999999E+09]];
	LOCAL CONST Robtarget Tr_meulage_bavure_App1 :=[[-142.68400198945,-248.862617015023,40.7135956821049],[0.673408716447437,-0.735943323251172,0.0516857249855686,-0.0472938834031763],[0,0,0,0],[8.999999E+09,8.999999E+09,8.999999E+09,8.999999E+09,8.999999E+09,8.999999E+09]];
	LOCAL CONST Robtarget Tr_meulage_bavure_App2 :=[[-116.231732521347,-61.4670496007511,23.8856797841052],[0.673408716447437,-0.735943323251172,0.0516857249855686,-0.0472938834031763],[0,0,0,0],[8.999999E+09,8.999999E+09,8.999999E+09,8.999999E+09,8.999999E+09,8.999999E+09]];
	LOCAL CONST Robtarget Tr_meulage_bavure_P0 :=[[-114.8395078125,-51.604125,23],[0.673408716447437,-0.735943323251172,0.0516857249855686,-0.0472938834031763],[0,0,0,0],[8.999999E+09,8.999999E+09,8.999999E+09,8.999999E+09,8.999999E+09,8.999999E+09]];
	LOCAL CONST Robtarget Tr_meulage_bavure_P1 :=[[-117.9325859375,-50.9020859375,23],[0.673553825642929,-0.735968958725782,0.0504388121725264,-0.0461612606033138],[0,0,0,0],[8.999999E+09,8.999999E+09,8.999999E+09,8.999999E+09,8.999999E+09,8.999999E+09]];
	LOCAL CONST Robtarget Tr_meulage_bavure_P2 :=[[-118.9293203125,-50.72306640625,23],[0.673960807585343,-0.736022323081527,0.0469235007904708,-0.0429669039861094],[0,0,0,0],[8.999999E+09,8.999999E+09,8.999999E+09,8.999999E+09,8.999999E+09,8.999999E+09]];
	LOCAL CONST Robtarget Tr_meulage_bavure_P3 :=[[-125.1540234375,-49.67340234375,23],[0.674565241671654,-0.736041788404539,0.0417311709212143,-0.0382456510502338],[0,0,0,0],[8.999999E+09,8.999999E+09,8.999999E+09,8.999999E+09,8.999999E+09,8.999999E+09]];
	LOCAL CONST Robtarget Tr_meulage_bavure_P4 :=[[-125.788390625,-49.5876171875,23],[0.675291409237207,-0.735970382369754,0.0355599861309368,-0.0326281515154118],[0,0,0,0],[8.999999E+09,8.999999E+09,8.999999E+09,8.999999E+09,8.999999E+09,8.999999E+09]];
	LOCAL CONST Robtarget Tr_meulage_bavure_P5 :=[[-128.6767578125,-49.35108984375,23],[0.676087857390827,-0.735769173434973,0.0289797372245318,-0.0266290694898412],[0,0,0,0],[8.999999E+09,8.999999E+09,8.999999E+09,8.999999E+09,8.999999E+09,8.999999E+09]];
	LOCAL CONST Robtarget Tr_meulage_bavure_P6 :=[[-129.0750390625,-49.33221484375,23],[0.676924092300665,-0.735431450803674,0.0222483662920997,-0.0204783942011106],[0,0,0,0],[8.999999E+09,8.999999E+09,8.999999E+09,8.999999E+09,8.999999E+09,8.999999E+09]];
	LOCAL CONST Robtarget Tr_meulage_bavure_P7 :=[[-130.4560546875,-49.3076796875,23],[0.677776237574307,-0.734973254291515,0.0153092551036926,-0.0141178597502141],[0,0,0,0],[8.999999E+09,8.999999E+09,8.999999E+09,8.999999E+09,8.999999E+09,8.999999E+09]];
	LOCAL CONST Robtarget Tr_meulage_bavure_P8 :=[[-136.033265625,-49.21208203125,23],[0.678627072761392,-0.734403926974957,0.00791596328148083,-0.00731475798601112],[0,0,0,0],[8.999999E+09,8.999999E+09,8.999999E+09,8.999999E+09,8.999999E+09,8.999999E+09]];
	LOCAL CONST Robtarget Tr_meulage_bavure_P9 :=[[-136.401546875,-49.2046953125,23],[0.679446184572836,-0.733725289189824,-0.000210456065891988,0.000194887068903422],[0,0,0,0],[8.999999E+09,8.999999E+09,8.999999E+09,8.999999E+09,8.999999E+09,8.999999E+09]];
	LOCAL CONST Robtarget Tr_meulage_bavure_P10 :=[[-140.495296875,-49.1396171875,23],[0.680191588202764,-0.732927027757378,-0.00919524336478197,0.00853362879431487],[0,0,0,0],[8.999999E+09,8.999999E+09,8.999999E+09,8.999999E+09,8.999999E+09,8.999999E+09]];
	LOCAL CONST Robtarget Tr_meulage_bavure_P11 :=[[-141.395453125,-49.1530625,23],[0.68082444531834,-0.731989466314166,-0.0189462911913733,0.0176219724255844],[0,0,0,0],[8.999999E+09,8.999999E+09,8.999999E+09,8.999999E+09,8.999999E+09,8.999999E+09]];
	LOCAL CONST Robtarget Tr_meulage_bavure_P12 :=[[-150.408328125,-49.87324609375,23],[0.681303639121852,-0.73091254594213,-0.0291884107438632,0.0272073185367814],[0,0,0,0],[8.999999E+09,8.999999E+09,8.999999E+09,8.999999E+09,8.999999E+09,8.999999E+09]];
	LOCAL CONST Robtarget Tr_meulage_bavure_P13 :=[[-150.415453125,-49.8739453125,23],[0.681619050335453,-0.72969693155302,-0.0396092691733578,0.0369995148272921],[0,0,0,0],[8.999999E+09,8.999999E+09,8.999999E+09,8.999999E+09,8.999999E+09,8.999999E+09]];
	LOCAL CONST Robtarget Tr_meulage_bavure_P14 :=[[-150.42959375,-49.8759921875,23],[0.681767406839203,-0.728356649377844,-0.049996748010429,0.0467987122388178],[0,0,0,0],[8.999999E+09,8.999999E+09,8.999999E+09,8.999999E+09,8.999999E+09,8.999999E+09]];
	LOCAL CONST Robtarget Tr_meulage_bavure_P15 :=[[-155.7309375,-50.50767578125,23],[0.681739357544111,-0.726909926441466,-0.0602959579086233,0.0565491350604657],[0,0,0,0],[8.999999E+09,8.999999E+09,8.999999E+09,8.999999E+09,8.999999E+09,8.999999E+09]];
	LOCAL CONST Robtarget Tr_meulage_bavure_P16 :=[[-157.44825,-50.75971875,23],[0.681528125365933,-0.725354837140657,-0.0705818628922506,0.0663172315654702],[0,0,0,0],[8.999999E+09,8.999999E+09,8.999999E+09,8.999999E+09,8.999999E+09,8.999999E+09]];
	LOCAL CONST Robtarget Tr_meulage_bavure_P17 :=[[-159.665796875,-51.17297265625,23],[0.681115173289887,-0.723684762714583,-0.0809661571545686,0.0762034534955382],[0,0,0,0],[8.999999E+09,8.999999E+09,8.999999E+09,8.999999E+09,8.999999E+09,8.999999E+09]];
	LOCAL CONST Robtarget Tr_meulage_bavure_P18 :=[[-163.16365625,-52.00669921875,23],[0.680485181273776,-0.721888810357199,-0.0915138769695578,0.0862651370477426],[0,0,0,0],[8.999999E+09,8.999999E+09,8.999999E+09,8.999999E+09,8.999999E+09,8.999999E+09]];
	LOCAL CONST Robtarget Tr_meulage_bavure_P19 :=[[-164.35084375,-52.3565234375,23],[0.679625010249021,-0.719957670656034,-0.102248099245485,0.0965200710124181],[0,0,0,0],[8.999999E+09,8.999999E+09,8.999999E+09,8.999999E+09,8.999999E+09,8.999999E+09]];
	LOCAL CONST Robtarget Tr_meulage_bavure_P20 :=[[-166.020234375,-52.86316015625,23],[0.678526555321443,-0.717897105732262,-0.113115852017145,0.106912409603819],[0,0,0,0],[8.999999E+09,8.999999E+09,8.999999E+09,8.999999E+09,8.999999E+09,8.999999E+09]];
	LOCAL CONST Robtarget Tr_meulage_bavure_P21 :=[[-170.21984375,-54.2692578125,23],[0.677226279368229,-0.715741131037852,-0.123866908634193,0.117201488126777],[0,0,0,0],[8.999999E+09,8.999999E+09,8.999999E+09,8.999999E+09,8.999999E+09,8.999999E+09]];
	LOCAL CONST Robtarget Tr_meulage_bavure_P22 :=[[-173.925578125,-55.6301875,23],[0.675825165804368,-0.71359117168927,-0.133973036024765,0.126882664580074],[0,0,0,0],[8.999999E+09,8.999999E+09,8.999999E+09,8.999999E+09,8.999999E+09,8.999999E+09]];
	LOCAL CONST Robtarget Tr_meulage_bavure_P23 :=[[-175.873390625,-56.41711328125,23],[0.674517564197697,-0.711669503126492,-0.142508993973569,0.135069465628389],[0,0,0,0],[8.999999E+09,8.999999E+09,8.999999E+09,8.999999E+09,8.999999E+09,8.999999E+09]];
	LOCAL CONST Robtarget Tr_meulage_bavure_P24 :=[[-179.0630625,-57.874421875,23],[0.673614327462585,-0.710299569289977,-0.148203355446694,0.14054901329409],[0,0,0,0],[8.999999E+09,8.999999E+09,8.999999E+09,8.999999E+09,8.999999E+09,8.999999E+09]];
	LOCAL CONST Robtarget Tr_meulage_bavure_P25 :=[[-179.64996875,-58.1318984375,23],[0.67345278923325,-0.709829312868415,-0.149737869163259,0.14206427350026],[0,0,0,0],[8.999999E+09,8.999999E+09,8.999999E+09,8.999999E+09,8.999999E+09,8.999999E+09]];
	LOCAL CONST Robtarget Tr_meulage_bavure_P26 :=[[-179.973640625,-58.3098125,23],[0.674248963492418,-0.710500395494755,-0.146117471128881,0.138662207764399],[0,0,0,0],[8.999999E+09,8.999999E+09,8.999999E+09,8.999999E+09,8.999999E+09,8.999999E+09]];
	LOCAL CONST Robtarget Tr_meulage_bavure_P27 :=[[-181.070703125,-58.91941796875,23],[0.676011419867312,-0.712303379056818,-0.136919906214186,0.129943817380891],[0,0,0,0],[8.999999E+09,8.999999E+09,8.999999E+09,8.999999E+09,8.999999E+09,8.999999E+09]];
	LOCAL CONST Robtarget Tr_meulage_bavure_P28 :=[[-185.38584375,-61.31100390625,23],[0.678502826176453,-0.714961938554709,-0.122376003587847,0.116135502902971],[0,0,0,0],[8.999999E+09,8.999999E+09,8.999999E+09,8.999999E+09,8.999999E+09,8.999999E+09]];
	LOCAL CONST Robtarget Tr_meulage_bavure_P29 :=[[-187.453421875,-62.6051484375,23],[0.681333993561771,-0.718066970881809,-0.103008855303411,0.0977393998082272],[0,0,0,0],[8.999999E+09,8.999999E+09,8.999999E+09,8.999999E+09,8.999999E+09,8.999999E+09]];
	LOCAL CONST Robtarget Tr_meulage_bavure_P30 :=[[-188.04903125,-62.747328125,23],[0.684123125450688,-0.721194225956988,-0.0789918449561947,0.0749314760317716],[0,0,0,0],[8.999999E+09,8.999999E+09,8.999999E+09,8.999999E+09,8.999999E+09,8.999999E+09]];
	LOCAL CONST Robtarget Tr_meulage_bavure_P31 :=[[-190.934890625,-63.2366640625,23],[0.686484621023572,-0.723914879519924,-0.0496722482962312,0.0471039282541623],[0,0,0,0],[8.999999E+09,8.999999E+09,8.999999E+09,8.999999E+09,8.999999E+09,8.999999E+09]];
	LOCAL CONST Robtarget Tr_meulage_bavure_P32 :=[[-192.509484375,-62.92959765625,23],[0.687859739840905,-0.725599664119422,-0.0136565330620622,0.0129462288142029],[0,0,0,0],[8.999999E+09,8.999999E+09,8.999999E+09,8.999999E+09,8.999999E+09,8.999999E+09]];
	LOCAL CONST Robtarget Tr_meulage_bavure_P33 :=[[-192.95103125,-62.7920546875,23],[0.687300790663922,-0.725182040178744,0.0301768549683229,-0.0286005101206955],[0,0,0,0],[8.999999E+09,8.999999E+09,8.999999E+09,8.999999E+09,8.999999E+09,8.999999E+09]];
	LOCAL CONST Robtarget Tr_meulage_bavure_P34 :=[[-192.971984375,-62.78340234375,23],[0.68353817883561,-0.721294105424518,0.0811860133281081,-0.0769363554753545],[0,0,0,0],[8.999999E+09,8.999999E+09,8.999999E+09,8.999999E+09,8.999999E+09,8.999999E+09]];
	LOCAL CONST Robtarget Tr_meulage_bavure_P35 :=[[-193.579015625,-62.24717578125,23],[0.675723630336173,-0.713002267314711,0.135838898246412,-0.128736692254328],[0,0,0,0],[8.999999E+09,8.999999E+09,8.999999E+09,8.999999E+09,8.999999E+09,8.999999E+09]];
	LOCAL CONST Robtarget Tr_meulage_bavure_P36 :=[[-194.635203125,-61.38554296875,23],[0.664361378958713,-0.700766341328822,0.188614394448454,-0.178815836031199],[0,0,0,0],[8.999999E+09,8.999999E+09,8.999999E+09,8.999999E+09,8.999999E+09,8.999999E+09]];
	LOCAL CONST Robtarget Tr_meulage_bavure_P37 :=[[-195.088484375,-60.98025390625,23],[0.651272123437156,-0.686474738127479,0.234625401936936,-0.222593746346116],[0,0,0,0],[8.999999E+09,8.999999E+09,8.999999E+09,8.999999E+09,8.999999E+09,8.999999E+09]];
	LOCAL CONST Robtarget Tr_meulage_bavure_P38 :=[[-195.48475,-60.71115234375,23],[0.638587712274317,-0.672319234823155,0.271479760025012,-0.257859109041785],[0,0,0,0],[8.999999E+09,8.999999E+09,8.999999E+09,8.999999E+09,8.999999E+09,8.999999E+09]];
	LOCAL CONST Robtarget Tr_meulage_bavure_P39 :=[[-197.147546875,-58.15252734375,23],[0.627839052693838,-0.65988009356052,0.299039925414476,-0.284519786734014],[0,0,0,0],[8.999999E+09,8.999999E+09,8.999999E+09,8.999999E+09,8.999999E+09,8.999999E+09]];
	LOCAL CONST Robtarget Tr_meulage_bavure_P40 :=[[-197.43440625,-57.7379296875,23],[0.619773638291652,-0.649884518439377,0.31835910472862,-0.303608679730898],[0,0,0,0],[8.999999E+09,8.999999E+09,8.999999E+09,8.999999E+09,8.999999E+09,8.999999E+09]];
	LOCAL CONST Robtarget Tr_meulage_bavure_P41 :=[[-198.2588125,-56.300078125,23],[0.614526624961947,-0.64241131843143,0.330879747412133,-0.316517484377329],[0,0,0,0],[8.999999E+09,8.999999E+09,8.999999E+09,8.999999E+09,8.999999E+09,8.999999E+09]];
	LOCAL CONST Robtarget Tr_meulage_bavure_P42 :=[[-199.957,-53.2754375,23],[0.611802670896982,-0.637106606381401,0.338153346824775,-0.324722924998679],[0,0,0,0],[8.999999E+09,8.999999E+09,8.999999E+09,8.999999E+09,8.999999E+09,8.999999E+09]];
	LOCAL CONST Robtarget Tr_meulage_bavure_P43 :=[[-201.824671875,-50.3134609375,23],[0.611092178805599,-0.633371920047636,0.341668487242838,-0.329649821360467],[0,0,0,0],[8.999999E+09,8.999999E+09,8.999999E+09,8.999999E+09,8.999999E+09,8.999999E+09]];
	LOCAL CONST Robtarget Tr_meulage_bavure_P44 :=[[-203.043671875,-48.44674609375,23],[0.611798690717634,-0.630534981343199,0.34278817979337,-0.332602259662602],[0,0,0,0],[8.999999E+09,8.999999E+09,8.999999E+09,8.999999E+09,8.999999E+09,8.999999E+09]];
	LOCAL CONST Robtarget Tr_meulage_bavure_P45 :=[[-204.021265625,-46.9410390625,23],[0.613361139921035,-0.627990908189829,0.342653078878095,-0.33467058251517],[0,0,0,0],[8.999999E+09,8.999999E+09,8.999999E+09,8.999999E+09,8.999999E+09,8.999999E+09]];
	LOCAL CONST Robtarget Tr_meulage_bavure_P46 :=[[-206.4303125,-43.3107890625,23],[0.615389814124426,-0.625326378641327,0.342016285239092,-0.336581576261209],[0,0,0,0],[8.999999E+09,8.999999E+09,8.999999E+09,8.999999E+09,8.999999E+09,8.999999E+09]];
	LOCAL CONST Robtarget Tr_meulage_bavure_P47 :=[[-209.07,-39.27465625,23],[0.617631242619502,-0.622306242316665,0.341328636810083,-0.338764447082884],[0,0,0,0],[8.999999E+09,8.999999E+09,8.999999E+09,8.999999E+09,8.999999E+09,8.999999E+09]];
	LOCAL CONST Robtarget Tr_meulage_bavure_P48 :=[[-213.2116875,-32.69418359375,23],[0.619955502730683,-0.618789697285662,0.340819884006908,-0.341461991783249],[0,0,0,0],[8.999999E+09,8.999999E+09,8.999999E+09,8.999999E+09,8.999999E+09,8.999999E+09]];
	LOCAL CONST Robtarget Tr_meulage_bavure_P49 :=[[-213.96253125,-31.5485234375,23],[0.622265048654706,-0.614755122100708,0.340595628442473,-0.344756387844486],[0,0,0,0],[8.999999E+09,8.999999E+09,8.999999E+09,8.999999E+09,8.999999E+09,8.999999E+09]];
	LOCAL CONST Robtarget Tr_meulage_bavure_P50 :=[[-216.67834375,-27.404509765625,23],[0.624537187030411,-0.610247143699464,0.340627460882325,-0.348603870482885],[0,0,0,0],[8.999999E+09,8.999999E+09,8.999999E+09,8.999999E+09,8.999999E+09,8.999999E+09]];
	LOCAL CONST Robtarget Tr_meulage_bavure_P51 :=[[-217.834203125,-25.641265625,23],[0.626858864702077,-0.605394339698564,0.340711099053136,-0.35279116228637],[0,0,0,0],[8.999999E+09,8.999999E+09,8.999999E+09,8.999999E+09,8.999999E+09,8.999999E+09]];
	LOCAL CONST Robtarget Tr_meulage_bavure_P52 :=[[-218.84184375,-24.062224609375,23],[0.629419108807383,-0.600480518776697,0.34045107825473,-0.356858228646868],[0,0,0,0],[8.999999E+09,8.999999E+09,8.999999E+09,8.999999E+09,8.999999E+09,8.999999E+09]];
	LOCAL CONST Robtarget Tr_meulage_bavure_P53 :=[[-220.044859375,-22.194548828125,23],[0.632522040486419,-0.595874602055739,0.339302863821293,-0.360170645009392],[0,0,0,0],[8.999999E+09,8.999999E+09,8.999999E+09,8.999999E+09,8.999999E+09,8.999999E+09]];
	LOCAL CONST Robtarget Tr_meulage_bavure_P54 :=[[-220.39490625,-21.54425,23],[0.636478219971316,-0.591933371593448,0.3367496863205,-0.362091159598246],[0,0,0,0],[8.999999E+09,8.999999E+09,8.999999E+09,8.999999E+09,8.999999E+09,8.999999E+09]];
	LOCAL CONST Robtarget Tr_meulage_bavure_P55 :=[[-221.3815,-19.6484375,23],[0.641440809211903,-0.588873120292858,0.332534592556579,-0.362219382732844],[0,0,0,0],[8.999999E+09,8.999999E+09,8.999999E+09,8.999999E+09,8.999999E+09,8.999999E+09]];
	LOCAL CONST Robtarget Tr_meulage_bavure_P56 :=[[-222.68240625,-17.3473515625,23],[0.647304248321752,-0.5866493890309,0.32681199958514,-0.360601748999426],[0,0,0,0],[8.999999E+09,8.999999E+09,8.999999E+09,8.999999E+09,8.999999E+09,8.999999E+09]];
	LOCAL CONST Robtarget Tr_meulage_bavure_P57 :=[[-223.70109375,-15.2891845703125,23],[0.653640019477949,-0.584968673808249,0.320217465056932,-0.357808818606247],[0,0,0,0],[8.999999E+09,8.999999E+09,8.999999E+09,8.999999E+09,8.999999E+09,8.999999E+09]];
	LOCAL CONST Robtarget Tr_meulage_bavure_P58 :=[[-225.889140625,-12.786041015625,23],[0.659833646308829,-0.583365988806962,0.313699222406597,-0.354818939973004],[0,0,0,0],[8.999999E+09,8.999999E+09,8.999999E+09,8.999999E+09,8.999999E+09,8.999999E+09]];
	LOCAL CONST Robtarget Tr_meulage_bavure_P59 :=[[-225.941765625,-12.714111328125,23],[0.665253145773851,-0.581393610185883,0.308247311585726,-0.352708543946972],[0,0,0,0],[8.999999E+09,8.999999E+09,8.999999E+09,8.999999E+09,8.999999E+09,8.999999E+09]];
	LOCAL CONST Robtarget Tr_meulage_bavure_P60 :=[[-226.1988125,-12.412689453125,23],[0.669422935290264,-0.578749134525273,0.304607168672559,-0.352330591613759],[0,0,0,0],[8.999999E+09,8.999999E+09,8.999999E+09,8.999999E+09,8.999999E+09,8.999999E+09]];
	LOCAL CONST Robtarget Tr_meulage_bavure_P61 :=[[-228.002859375,-10.0315546875,23],[0.672093919747293,-0.575345701460376,0.303123108161059,-0.354095281172408],[0,0,0,0],[8.999999E+09,8.999999E+09,8.999999E+09,8.999999E+09,8.999999E+09,8.999999E+09]];
	LOCAL CONST Robtarget Tr_meulage_bavure_P62 :=[[-229.053921875,-8.2217099609375,23],[0.673250679230681,-0.57128247293793,0.303726500662445,-0.357938642541842],[0,0,0,0],[8.999999E+09,8.999999E+09,8.999999E+09,8.999999E+09,8.999999E+09,8.999999E+09]];
	LOCAL CONST Robtarget Tr_meulage_bavure_P63 :=[[-229.846671875,-7.2158203125,23],[0.673058934923327,-0.566800979741563,0.306039109048894,-0.363412139610718],[0,0,0,0],[8.999999E+09,8.999999E+09,8.999999E+09,8.999999E+09,8.999999E+09,8.999999E+09]];
	LOCAL CONST Robtarget Tr_meulage_bavure_P64 :=[[-231.171078125,-5.173431640625,23],[0.671853761138813,-0.562270314954965,0.30943852473915,-0.369746421174476],[0,0,0,0],[8.999999E+09,8.999999E+09,8.999999E+09,8.999999E+09,8.999999E+09,8.999999E+09]];
	LOCAL CONST Robtarget Tr_meulage_bavure_P65 :=[[-232.326015625,-3.03558349609375,23],[0.670115275942213,-0.558150930204681,0.313149076288066,-0.375966370943561],[0,0,0,0],[8.999999E+09,8.999999E+09,8.999999E+09,8.999999E+09,8.999999E+09,8.999999E+09]];
	LOCAL CONST Robtarget Tr_meulage_bavure_P66 :=[[-232.51621875,-2.6107177734375,23],[0.668380295050204,-0.554945581592507,0.316384887087642,-0.381056145314698],[0,0,0,0],[8.999999E+09,8.999999E+09,8.999999E+09,8.999999E+09,8.999999E+09,8.999999E+09]];
	LOCAL CONST Robtarget Tr_meulage_bavure_P67 :=[[-235.38821875,1.14218139648438,23],[0.667080662526292,-0.553063158169367,0.318565704996245,-0.384240060846672],[0,0,0,0],[8.999999E+09,8.999999E+09,8.999999E+09,8.999999E+09,8.999999E+09,8.999999E+09]];
	LOCAL CONST Robtarget Tr_meulage_bavure_P68 :=[[-235.4095,1.17611694335938,23],[0.666357636060518,-0.552628837823808,0.319544417640668,-0.385305377102413],[0,0,0,0],[8.999999E+09,8.999999E+09,8.999999E+09,8.999999E+09,8.999999E+09,8.999999E+09]];
	LOCAL CONST Robtarget Tr_meulage_bavure_P69 :=[[-235.442921875,1.22854614257813,23],[0.665977793569522,-0.553495068585247,0.319660048665835,-0.384622205301566],[0,0,0,0],[8.999999E+09,8.999999E+09,8.999999E+09,8.999999E+09,8.999999E+09,8.999999E+09]];
	LOCAL CONST Robtarget Tr_meulage_bavure_P70 :=[[-237.888171875,5.9194033203125,23],[0.665492090183466,-0.555299141832911,0.319544667178807,-0.382954757981226],[0,0,0,0],[8.999999E+09,8.999999E+09,8.999999E+09,8.999999E+09,8.999999E+09,8.999999E+09]];
	LOCAL CONST Robtarget Tr_meulage_bavure_P71 :=[[-238.607265625,7.010345703125,23],[0.664462262579911,-0.557666346387545,0.31982074211143,-0.381068026248918],[0,0,0,0],[8.999999E+09,8.999999E+09,8.999999E+09,8.999999E+09,8.999999E+09,8.999999E+09]];
	LOCAL CONST Robtarget Tr_meulage_bavure_P72 :=[[-239.614640625,8.508208984375,23],[0.662639995830684,-0.560409687033395,0.32083411874636,-0.379360892624543],[0,0,0,0],[8.999999E+09,8.999999E+09,8.999999E+09,8.999999E+09,8.999999E+09,8.999999E+09]];
	LOCAL CONST Robtarget Tr_meulage_bavure_P73 :=[[-241.36415625,11.366302734375,23],[0.660113882782712,-0.563520053174085,0.322480830472116,-0.377757760219724],[0,0,0,0],[8.999999E+09,8.999999E+09,8.999999E+09,8.999999E+09,8.999999E+09,8.999999E+09]];
	LOCAL CONST Robtarget Tr_meulage_bavure_P74 :=[[-242.08009375,12.827576171875,23],[0.657157367207894,-0.567181933592564,0.324361587353777,-0.375816989477494],[0,0,0,0],[8.999999E+09,8.999999E+09,8.999999E+09,8.999999E+09,8.999999E+09,8.999999E+09]];
	LOCAL CONST Robtarget Tr_meulage_bavure_P75 :=[[-243.048765625,14.4635009765625,23],[0.654070697774336,-0.571619761954739,0.326013658356217,-0.373038154376998],[0,0,0,0],[8.999999E+09,8.999999E+09,8.999999E+09,8.999999E+09,8.999999E+09,8.999999E+09]];
	LOCAL CONST Robtarget Tr_meulage_bavure_P76 :=[[-243.74178125,15.730712890625,23],[0.651061406576409,-0.576897577676238,0.327127917961487,-0.369182278865358],[0,0,0,0],[8.999999E+09,8.999999E+09,8.999999E+09,8.999999E+09,8.999999E+09,8.999999E+09]];
	LOCAL CONST Robtarget Tr_meulage_bavure_P77 :=[[-243.966125,15.999451171875,23],[0.648092361501352,-0.582894332963311,0.327747334308964,-0.364406603145753],[0,0,0,0],[8.999999E+09,8.999999E+09,8.999999E+09,8.999999E+09,8.999999E+09,8.999999E+09]];
	LOCAL CONST Robtarget Tr_meulage_bavure_P78 :=[[-246.559359375,20.1897578125,23],[0.644953286748676,-0.589299372348973,0.328217244013777,-0.359214348813054],[0,0,0,0],[8.999999E+09,8.999999E+09,8.999999E+09,8.999999E+09,8.999999E+09,8.999999E+09]];
	LOCAL CONST Robtarget Tr_meulage_bavure_P79 :=[[-247.57825,21.1435546875,23],[0.641379706580527,-0.595722496822702,0.329026336399039,-0.354243487903208],[0,0,0,0],[8.999999E+09,8.999999E+09,8.999999E+09,8.999999E+09,8.999999E+09,8.999999E+09]];
	LOCAL CONST Robtarget Tr_meulage_bavure_P80 :=[[-248.749546875,22.633025390625,23],[0.63710672764735,-0.601738919048275,0.330733305968345,-0.35017248780044],[0,0,0,0],[8.999999E+09,8.999999E+09,8.999999E+09,8.999999E+09,8.999999E+09,8.999999E+09]];
	LOCAL CONST Robtarget Tr_meulage_bavure_P81 :=[[-250.58128125,25.4924921875,23],[0.631901145349445,-0.606908732557199,0.333909364410898,-0.347659703173354],[0,0,0,0],[8.999999E+09,8.999999E+09,8.999999E+09,8.999999E+09,8.999999E+09,8.999999E+09]];
	LOCAL CONST Robtarget Tr_meulage_bavure_P82 :=[[-251.363265625,26.859283203125,23],[0.625411651044696,-0.610718047534943,0.339320444899579,-0.347484343281544],[0,0,0,0],[8.999999E+09,8.999999E+09,8.999999E+09,8.999999E+09,8.999999E+09,8.999999E+09]];
	LOCAL CONST Robtarget Tr_meulage_bavure_P83 :=[[-251.812859375,27.59881640625,23],[0.617127863171467,-0.612431679274201,0.34800587715891,-0.35067441905799],[0,0,0,0],[8.999999E+09,8.999999E+09,8.999999E+09,8.999999E+09,8.999999E+09,8.999999E+09]];
	LOCAL CONST Robtarget Tr_meulage_bavure_P84 :=[[-253.3178125,29.85269140625,23],[0.606366200716965,-0.611092722828723,0.361175733209593,-0.358382204461053],[0,0,0,0],[8.999999E+09,8.999999E+09,8.999999E+09,8.999999E+09,8.999999E+09,8.999999E+09]];
	LOCAL CONST Robtarget Tr_meulage_bavure_P85 :=[[-254.989203125,32.302978515625,23],[0.592246468803047,-0.605595749863351,0.379995847434239,-0.371619514921515],[0,0,0,0],[8.999999E+09,8.999999E+09,8.999999E+09,8.999999E+09,8.999999E+09,8.999999E+09]];
	LOCAL CONST Robtarget Tr_meulage_bavure_P86 :=[[-255.835703125,33.5635390625,23],[0.573934318699078,-0.594854015088483,0.405020477222017,-0.390776805329315],[0,0,0,0],[8.999999E+09,8.999999E+09,8.999999E+09,8.999999E+09,8.999999E+09,8.999999E+09]];
	LOCAL CONST Robtarget Tr_meulage_bavure_P87 :=[[-256.98275,35.17178515625,23],[0.550796235120078,-0.57797912269148,0.435898987719791,-0.415398259042088],[0,0,0,0],[8.999999E+09,8.999999E+09,8.999999E+09,8.999999E+09,8.999999E+09,8.999999E+09]];
	LOCAL CONST Robtarget Tr_meulage_bavure_P88 :=[[-257.62634375,37.013,23],[0.522490840491545,-0.554415322617577,0.471425761566886,-0.444280005154821],[0,0,0,0],[8.999999E+09,8.999999E+09,8.999999E+09,8.999999E+09,8.999999E+09,8.999999E+09]];
	LOCAL CONST Robtarget Tr_meulage_bavure_P89 :=[[-258.0756875,38.17721484375,23],[0.488849753538399,-0.523858595684437,0.510000420861065,-0.475917703930535],[0,0,0,0],[8.999999E+09,8.999999E+09,8.999999E+09,8.999999E+09,8.999999E+09,8.999999E+09]];
	LOCAL CONST Robtarget Tr_meulage_bavure_P90 :=[[-257.89328125,40.1533828125,23],[0.449709803341687,-0.48610633112542,0.550031555172177,-0.508848716155442],[0,0,0,0],[8.999999E+09,8.999999E+09,8.999999E+09,8.999999E+09,8.999999E+09,8.999999E+09]];
	LOCAL CONST Robtarget Tr_meulage_bavure_P91 :=[[-257.800421875,41.47079296875,23],[0.405389346883589,-0.44148405579803,0.58960638042099,-0.541401534977763],[0,0,0,0],[8.999999E+09,8.999999E+09,8.999999E+09,8.999999E+09,8.999999E+09,8.999999E+09]];
	LOCAL CONST Robtarget Tr_meulage_bavure_P92 :=[[-256.7125,42.755859375,23],[0.357695503734552,-0.392020282813091,0.626105463162067,-0.571284494336965],[0,0,0,0],[8.999999E+09,8.999999E+09,8.999999E+09,8.999999E+09,8.999999E+09,8.999999E+09]];
	LOCAL CONST Robtarget Tr_meulage_bavure_P93 :=[[-255.583171875,44.17044140625,23],[0.310516678401752,-0.342142820350356,0.656720725823948,-0.596016418557671],[0,0,0,0],[8.999999E+09,8.999999E+09,8.999999E+09,8.999999E+09,8.999999E+09,8.999999E+09]];
	LOCAL CONST Robtarget Tr_meulage_bavure_P94 :=[[-254.700328125,44.71005078125,23],[0.268612191448391,-0.297301996224077,0.679836707060288,-0.614232094065343],[0,0,0,0],[8.999999E+09,8.999999E+09,8.999999E+09,8.999999E+09,8.999999E+09,8.999999E+09]];
	LOCAL CONST Robtarget Tr_meulage_bavure_P95 :=[[-248.42134375,48.47122265625,23],[0.23520201813738,-0.26130502596738,0.695807489157552,-0.626299953776586],[0,0,0,0],[8.999999E+09,8.999999E+09,8.999999E+09,8.999999E+09,8.999999E+09,8.999999E+09]];
	LOCAL CONST Robtarget Tr_meulage_bavure_P96 :=[[-248.046484375,48.68933203125,23],[0.210909673263325,-0.235067637375651,0.706224696490845,-0.63364579510086],[0,0,0,0],[8.999999E+09,8.999999E+09,8.999999E+09,8.999999E+09,8.999999E+09,8.999999E+09]];
	LOCAL CONST Robtarget Tr_meulage_bavure_P97 :=[[-246.913,49.396453125,23],[0.194426057494722,-0.217291124927158,0.712846173682948,-0.637834937786046],[0,0,0,0],[8.999999E+09,8.999999E+09,8.999999E+09,8.999999E+09,8.999999E+09,8.999999E+09]];
	LOCAL CONST Robtarget Tr_meulage_bavure_P98 :=[[-244.058640625,51.13922265625,23],[0.183593030555603,-0.20569064299731,0.717128889011447,-0.640086802754103],[0,0,0,0],[8.999999E+09,8.999999E+09,8.999999E+09,8.999999E+09,8.999999E+09,8.999999E+09]];
	LOCAL CONST Robtarget Tr_meulage_bavure_P99 :=[[-241.151640625,52.8610859375,23],[0.176373374527833,-0.198052230838273,0.720056134358581,-0.641238574939332],[0,0,0,0],[8.999999E+09,8.999999E+09,8.999999E+09,8.999999E+09,8.999999E+09,8.999999E+09]];
	LOCAL CONST Robtarget Tr_meulage_bavure_P100 :=[[-239.340765625,53.87649609375,23],[0.17122666816448,-0.192685787584795,0.72224349196138,-0.641808346542447],[0,0,0,0],[8.999999E+09,8.999999E+09,8.999999E+09,8.999999E+09,8.999999E+09,8.999999E+09]];
	LOCAL CONST Robtarget Tr_meulage_bavure_P101 :=[[-235.800859375,55.82986328125,23],[0.167225101593044,-0.18859327818831,0.724065176417263,-0.642026448924981],[0,0,0,0],[8.999999E+09,8.999999E+09,8.999999E+09,8.999999E+09,8.999999E+09,8.999999E+09]];
	LOCAL CONST Robtarget Tr_meulage_bavure_P102 :=[[-233.68796875,56.9983203125,23],[0.16392425646201,-0.185286546141835,0.72568166604721,-0.642015462060808],[0,0,0,0],[8.999999E+09,8.999999E+09,8.999999E+09,8.999999E+09,8.999999E+09,8.999999E+09]];
	LOCAL CONST Robtarget Tr_meulage_bavure_P103 :=[[-231.82603125,58.03436328125,23],[0.161089361583765,-0.182508042041041,0.727176789189061,-0.641837167387156],[0,0,0,0],[8.999999E+09,8.999999E+09,8.999999E+09,8.999999E+09,8.999999E+09,8.999999E+09]];
	LOCAL CONST Robtarget Tr_meulage_bavure_P104 :=[[-229.550671875,59.1696796875,23],[0.158629552799477,-0.180164086339919,0.728592837163639,-0.641506075268021],[0,0,0,0],[8.999999E+09,8.999999E+09,8.999999E+09,8.999999E+09,8.999999E+09,8.999999E+09]];
	LOCAL CONST Robtarget Tr_meulage_bavure_P105 :=[[-226.269328125,60.95455859375,23],[0.15646083252117,-0.178164958110619,0.729963295169169,-0.641038878145461],[0,0,0,0],[8.999999E+09,8.999999E+09,8.999999E+09,8.999999E+09,8.999999E+09,8.999999E+09]];
	LOCAL CONST Robtarget Tr_meulage_bavure_P106 :=[[-223.00571875,62.6611640625,23],[0.154495972818499,-0.176411214197974,0.731312264517983,-0.640462684044622],[0,0,0,0],[8.999999E+09,8.999999E+09,8.999999E+09,8.999999E+09,8.999999E+09,8.999999E+09]];
	LOCAL CONST Robtarget Tr_meulage_bavure_P107 :=[[-220.135859375,64.2274765625,23],[0.152668772783652,-0.174819188086701,0.732644234873352,-0.639814756316453],[0,0,0,0],[8.999999E+09,8.999999E+09,8.999999E+09,8.999999E+09,8.999999E+09,8.999999E+09]];
	LOCAL CONST Robtarget Tr_meulage_bavure_P108 :=[[-219.192,64.732484375,23],[0.150901611471538,-0.173297776471793,0.733976311867266,-0.639120769450462],[0,0,0,0],[8.999999E+09,8.999999E+09,8.999999E+09,8.999999E+09,8.999999E+09,8.999999E+09]];
	LOCAL CONST Robtarget Tr_meulage_bavure_P109 :=[[-216.622984375,66.0360078125,23],[0.149115111754874,-0.171751376132187,0.735322647001926,-0.638409549622428],[0,0,0,0],[8.999999E+09,8.999999E+09,8.999999E+09,8.999999E+09,8.999999E+09,8.999999E+09]];
	LOCAL CONST Robtarget Tr_meulage_bavure_P110 :=[[-214.49690625,66.9835546875,23],[0.147259731822831,-0.170104645147006,0.736665851208285,-0.637732235931705],[0,0,0,0],[8.999999E+09,8.999999E+09,8.999999E+09,8.999999E+09,8.999999E+09,8.999999E+09]];
	LOCAL CONST Robtarget Tr_meulage_bavure_P111 :=[[-212.065578125,68.2174375,23],[0.145330159002698,-0.168344271333169,0.737995116672975,-0.637104825723677],[0,0,0,0],[8.999999E+09,8.999999E+09,8.999999E+09,8.999999E+09,8.999999E+09,8.999999E+09]];
	LOCAL CONST Robtarget Tr_meulage_bavure_P112 :=[[-210.58340625,68.8725,23],[0.143391964150477,-0.166535440093399,0.739273780161479,-0.636536699472798],[0,0,0,0],[8.999999E+09,8.999999E+09,8.999999E+09,8.999999E+09,8.999999E+09,8.999999E+09]];
	LOCAL CONST Robtarget Tr_meulage_bavure_P113 :=[[-208.288625,69.969296875,23],[0.141555544320676,-0.16479598526672,0.740452696837199,-0.636029963805611],[0,0,0,0],[8.999999E+09,8.999999E+09,8.999999E+09,8.999999E+09,8.999999E+09,8.999999E+09]];
	LOCAL CONST Robtarget Tr_meulage_bavure_P114 :=[[-207.481109375,70.3230625,23],[0.139926936614632,-0.163243701634301,0.741491029858451,-0.63558083587049],[0,0,0,0],[8.999999E+09,8.999999E+09,8.999999E+09,8.999999E+09,8.999999E+09,8.999999E+09]];
	LOCAL CONST Robtarget Tr_meulage_bavure_P115 :=[[-206.259203125,70.8953828125,23],[0.138577612985102,-0.161955518087636,0.742354806598105,-0.635197604262648],[0,0,0,0],[8.999999E+09,8.999999E+09,8.999999E+09,8.999999E+09,8.999999E+09,8.999999E+09]];
	LOCAL CONST Robtarget Tr_meulage_bavure_P116 :=[[-203.4735625,72.248203125,23],[0.13753515773138,-0.160957371958029,0.743021448250693,-0.634898363708407],[0,0,0,0],[8.999999E+09,8.999999E+09,8.999999E+09,8.999999E+09,8.999999E+09,8.999999E+09]];
	LOCAL CONST Robtarget Tr_meulage_bavure_P117 :=[[-199.53803125,74.02728125,23],[0.13679954933351,-0.160247556486764,0.743484300632692,-0.634694965046113],[0,0,0,0],[8.999999E+09,8.999999E+09,8.999999E+09,8.999999E+09,8.999999E+09,8.999999E+09]];
	LOCAL CONST Robtarget Tr_meulage_bavure_P118 :=[[-199.026484375,74.2523828125,23],[0.136385682078025,-0.15984174751313,0.743733734493427,-0.634594117253321],[0,0,0,0],[8.999999E+09,8.999999E+09,8.999999E+09,8.999999E+09,8.999999E+09,8.999999E+09]];
	LOCAL CONST Robtarget Tr_meulage_bavure_P119 :=[[-198.441,74.5859375,23],[0.136317560523005,-0.15977201022717,0.743769441626946,-0.634584466515661],[0,0,0,0],[8.999999E+09,8.999999E+09,8.999999E+09,8.999999E+09,8.999999E+09,8.999999E+09]];
	LOCAL CONST Robtarget Tr_meulage_bavure_P120 :=[[-197.18415625,75.163484375,23],[0.136608183934445,-0.160052201195074,0.743585416842907,-0.634667018863674],[0,0,0,0],[8.999999E+09,8.999999E+09,8.999999E+09,8.999999E+09,8.999999E+09,8.999999E+09]];
	LOCAL CONST Robtarget Tr_meulage_bavure_P121 :=[[-195.5825,75.822328125,23],[0.137204663683833,-0.160625400600039,0.743205287300173,-0.634838768408602],[0,0,0,0],[8.999999E+09,8.999999E+09,8.999999E+09,8.999999E+09,8.999999E+09,8.999999E+09]];
	LOCAL CONST Robtarget Tr_meulage_bavure_P122 :=[[-192.064359375,77.391171875,23],[0.137948791557134,-0.161310287107865,0.742677988141598,-0.635120876771542],[0,0,0,0],[8.999999E+09,8.999999E+09,8.999999E+09,8.999999E+09,8.999999E+09,8.999999E+09]];
	LOCAL CONST Robtarget Tr_meulage_bavure_P123 :=[[-190.5284375,77.9620078125,23],[0.138591202749135,-0.161832075425788,0.742098770596165,-0.63552519427918],[0,0,0,0],[8.999999E+09,8.999999E+09,8.999999E+09,8.999999E+09,8.999999E+09,8.999999E+09]];
	LOCAL CONST Robtarget Tr_meulage_bavure_P124 :=[[-189.0028125,78.63396875,23],[0.138864606150539,-0.161885620893695,0.741547341754122,-0.636095281262103],[0,0,0,0],[8.999999E+09,8.999999E+09,8.999999E+09,8.999999E+09,8.999999E+09,8.999999E+09]];
	LOCAL CONST Robtarget Tr_meulage_bavure_P125 :=[[-186.4945,79.5902734375,23],[0.138570473588223,-0.16125633110742,0.74109979240478,-0.636840417392695],[0,0,0,0],[8.999999E+09,8.999999E+09,8.999999E+09,8.999999E+09,8.999999E+09,8.999999E+09]];
	LOCAL CONST Robtarget Tr_meulage_bavure_P126 :=[[-185.92671875,79.8669140625,23],[0.137654929763961,-0.159900703846119,0.740795485295542,-0.637734219081066],[0,0,0,0],[8.999999E+09,8.999999E+09,8.999999E+09,8.999999E+09,8.999999E+09,8.999999E+09]];
	LOCAL CONST Robtarget Tr_meulage_bavure_P127 :=[[-181.411921875,81.77203125,23],[0.136222006047282,-0.157956635930949,0.740628796939654,-0.638719227342932],[0,0,0,0],[8.999999E+09,8.999999E+09,8.999999E+09,8.999999E+09,8.999999E+09,8.999999E+09]];
	LOCAL CONST Robtarget Tr_meulage_bavure_P128 :=[[-180.805546875,82.00271875,23],[0.134495025550458,-0.155698271452561,0.740564640730359,-0.639713333664994],[0,0,0,0],[8.999999E+09,8.999999E+09,8.999999E+09,8.999999E+09,8.999999E+09,8.999999E+09]];
	LOCAL CONST Robtarget Tr_meulage_bavure_P129 :=[[-180.6305,82.0803515625,23],[0.132744917037483,-0.153449580267774,0.74055471866643,-0.640633063443685],[0,0,0,0],[8.999999E+09,8.999999E+09,8.999999E+09,8.999999E+09,8.999999E+09,8.999999E+09]];
	LOCAL CONST Robtarget Tr_meulage_bavure_P130 :=[[-177.4739375,83.32171875,23],[0.131214302188678,-0.151492668177876,0.740548500756102,-0.641420841895067],[0,0,0,0],[8.999999E+09,8.999999E+09,8.999999E+09,8.999999E+09,8.999999E+09,8.999999E+09]];
	LOCAL CONST Robtarget Tr_meulage_bavure_P131 :=[[-173.523484375,84.9141875,23],[0.130048053978165,-0.150004655557617,0.740539488579928,-0.642018202873806],[0,0,0,0],[8.999999E+09,8.999999E+09,8.999999E+09,8.999999E+09,8.999999E+09,8.999999E+09]];
	LOCAL CONST Robtarget Tr_meulage_bavure_P132 :=[[-171.187109375,85.77865625,23],[0.12927138352539,-0.149007253511965,0.740515466772282,-0.642434892633706],[0,0,0,0],[8.999999E+09,8.999999E+09,8.999999E+09,8.999999E+09,8.999999E+09,8.999999E+09]];
	LOCAL CONST Robtarget Tr_meulage_bavure_P133 :=[[-170.139859375,86.17315625,23],[0.12877077706959,-0.148365037268687,0.740499071579657,-0.642702907787744],[0,0,0,0],[8.999999E+09,8.999999E+09,8.999999E+09,8.999999E+09,8.999999E+09,8.999999E+09]];
	LOCAL CONST Robtarget Tr_meulage_bavure_P134 :=[[-168.038953125,87.042359375,23],[0.128311713188016,-0.147809712564574,0.740551005396694,-0.642862817042858],[0,0,0,0],[8.999999E+09,8.999999E+09,8.999999E+09,8.999999E+09,8.999999E+09,8.999999E+09]];
	LOCAL CONST Robtarget Tr_meulage_bavure_P135 :=[[-165.92875,87.8045078125,23],[0.127618393794922,-0.147010575725101,0.740709020566689,-0.643002008582644],[0,0,0,0],[8.999999E+09,8.999999E+09,8.999999E+09,8.999999E+09,8.999999E+09,8.999999E+09]];
	LOCAL CONST Robtarget Tr_meulage_bavure_P136 :=[[-164.941484375,88.2270234375,23],[0.126459285733567,-0.145694976499326,0.741013502711612,-0.643179610741576],[0,0,0,0],[8.999999E+09,8.999999E+09,8.999999E+09,8.999999E+09,8.999999E+09,8.999999E+09]];
	LOCAL CONST Robtarget Tr_meulage_bavure_P137 :=[[-161.7071875,89.4457109375,23],[0.124748565307238,-0.143751563398004,0.741456252547539,-0.643440680274861],[0,0,0,0],[8.999999E+09,8.999999E+09,8.999999E+09,8.999999E+09,8.999999E+09,8.999999E+09]];
	LOCAL CONST Robtarget Tr_meulage_bavure_P138 :=[[-161.014625,89.6702890625,23],[0.122593626458139,-0.141294648370561,0.7419898178478,-0.643783919730735],[0,0,0,0],[8.999999E+09,8.999999E+09,8.999999E+09,8.999999E+09,8.999999E+09,8.999999E+09]];
	LOCAL CONST Robtarget Tr_meulage_bavure_P139 :=[[-159.9928125,90.055328125,23],[0.120263435815576,-0.138628419796378,0.742538810053031,-0.644169995261826],[0,0,0,0],[8.999999E+09,8.999999E+09,8.999999E+09,8.999999E+09,8.999999E+09,8.999999E+09]];
	LOCAL CONST Robtarget Tr_meulage_bavure_P140 :=[[-159.57665625,90.194734375,23],[0.118091651423145,-0.136130315843941,0.743013749161736,-0.64455679930399],[0,0,0,0],[8.999999E+09,8.999999E+09,8.999999E+09,8.999999E+09,8.999999E+09,8.999999E+09]];
	LOCAL CONST Robtarget Tr_meulage_bavure_P141 :=[[-158.5041875,90.609859375,23],[0.116339150267684,-0.134097970948062,0.743353376532998,-0.644909833929982],[0,0,0,0],[8.999999E+09,8.999999E+09,8.999999E+09,8.999999E+09,8.999999E+09,8.999999E+09]];
	LOCAL CONST Robtarget Tr_meulage_bavure_P142 :=[[-156.44215625,91.2901328125,23],[0.115087299838202,-0.132624713521047,0.743542323588631,-0.645221211532782],[0,0,0,0],[8.999999E+09,8.999999E+09,8.999999E+09,8.999999E+09,8.999999E+09,8.999999E+09]];
	LOCAL CONST Robtarget Tr_meulage_bavure_P143 :=[[-155.42975,91.6494140625,23],[0.114221064845451,-0.131574302874906,0.743598274100478,-0.645525644667464],[0,0,0,0],[8.999999E+09,8.999999E+09,8.999999E+09,8.999999E+09,8.999999E+09,8.999999E+09]];
	LOCAL CONST Robtarget Tr_meulage_bavure_P144 :=[[-151.36409375,92.919828125,23],[0.113471868480312,-0.130645652024638,0.743596480345916,-0.645848374688526],[0,0,0,0],[8.999999E+09,8.999999E+09,8.999999E+09,8.999999E+09,8.999999E+09,8.999999E+09]];
	LOCAL CONST Robtarget Tr_meulage_bavure_P145 :=[[-150.02296875,93.3269921875,23],[0.112537214085148,-0.129494771294398,0.743607519584635,-0.646230869326553],[0,0,0,0],[8.999999E+09,8.999999E+09,8.999999E+09,8.999999E+09,8.999999E+09,8.999999E+09]];
	LOCAL CONST Robtarget Tr_meulage_bavure_P146 :=[[-146.91446875,94.407015625,23],[0.111183487998567,-0.127866024857792,0.743706259987081,-0.64667573832607],[0,0,0,0],[8.999999E+09,8.999999E+09,8.999999E+09,8.999999E+09,8.999999E+09,8.999999E+09]];
	LOCAL CONST Robtarget Tr_meulage_bavure_P147 :=[[-145.930171875,94.703609375,23],[0.109326722180621,-0.125666697510076,0.743913344386977,-0.647185046951129],[0,0,0,0],[8.999999E+09,8.999999E+09,8.999999E+09,8.999999E+09,8.999999E+09,8.999999E+09]];
	LOCAL CONST Robtarget Tr_meulage_bavure_P148 :=[[-145.10603125,95.0021640625,23],[0.107017571032015,-0.122964133959389,0.744235479191889,-0.647719547923362],[0,0,0,0],[8.999999E+09,8.999999E+09,8.999999E+09,8.999999E+09,8.999999E+09,8.999999E+09]];
	LOCAL CONST Robtarget Tr_meulage_bavure_P149 :=[[-141.68346875,96.07165625,23],[0.104388527607819,-0.11992547976957,0.744682123500221,-0.648204789819631],[0,0,0,0],[8.999999E+09,8.999999E+09,8.999999E+09,8.999999E+09,8.999999E+09,8.999999E+09]];
	LOCAL CONST Robtarget Tr_meulage_bavure_P150 :=[[-138.10428125,97.3871796875,23],[0.1016084234248,-0.116751248320244,0.745241786658303,-0.648582726969453],[0,0,0,0],[8.999999E+09,8.999999E+09,8.999999E+09,8.999999E+09,8.999999E+09,8.999999E+09]];
	LOCAL CONST Robtarget Tr_meulage_bavure_P151 :=[[-137.86978125,97.45965625,23],[0.0988247800852614,-0.113613900211378,0.745903526980743,-0.64880927317475],[0,0,0,0],[8.999999E+09,8.999999E+09,8.999999E+09,8.999999E+09,8.999999E+09,8.999999E+09]];
	LOCAL CONST Robtarget Tr_meulage_bavure_P152 :=[[-137.494171875,97.5817578125,23],[0.0961469582082786,-0.110641580305925,0.746665705259689,-0.648848616954489],[0,0,0,0],[8.999999E+09,8.999999E+09,8.999999E+09,8.999999E+09,8.999999E+09,8.999999E+09]];
	LOCAL CONST Robtarget Tr_meulage_bavure_P153 :=[[-132.647859375,98.9463515625,23],[0.0936342150760023,-0.107901283109349,0.747526686141258,-0.648686211027432],[0,0,0,0],[8.999999E+09,8.999999E+09,8.999999E+09,8.999999E+09,8.999999E+09,8.999999E+09]];
	LOCAL CONST Robtarget Tr_meulage_bavure_P154 :=[[-126.50003125,100.6853359375,23],[0.0912778719722005,-0.105390028911929,0.748519634914639,-0.648289787087091],[0,0,0,0],[8.999999E+09,8.999999E+09,8.999999E+09,8.999999E+09,8.999999E+09,8.999999E+09]];
	LOCAL CONST Robtarget Tr_meulage_bavure_P155 :=[[-126.29828125,100.7319375,23],[0.0890146737456933,-0.103024567520216,0.749635251145542,-0.647695388732374],[0,0,0,0],[8.999999E+09,8.999999E+09,8.999999E+09,8.999999E+09,8.999999E+09,8.999999E+09]];
	LOCAL CONST Robtarget Tr_meulage_bavure_P156 :=[[-126.0548671875,100.809265625,23],[0.086751888538415,-0.100692341708716,0.750881592989009,-0.646925030792998],[0,0,0,0],[8.999999E+09,8.999999E+09,8.999999E+09,8.999999E+09,8.999999E+09,8.999999E+09]];
	LOCAL CONST Robtarget Tr_meulage_bavure_P157 :=[[-124.0311875,101.40634375,23],[0.0844240357571746,-0.0983124633251237,0.752263680089244,-0.645992722373871],[0,0,0,0],[8.999999E+09,8.999999E+09,8.999999E+09,8.999999E+09,8.999999E+09,8.999999E+09]];
	LOCAL CONST Robtarget Tr_meulage_bavure_P158 :=[[-117.3661796875,103.333859375,23],[0.0820781560406727,-0.0959254951276384,0.753739213237554,-0.644933077236324],[0,0,0,0],[8.999999E+09,8.999999E+09,8.999999E+09,8.999999E+09,8.999999E+09,8.999999E+09]];
	LOCAL CONST Robtarget Tr_meulage_bavure_P159 :=[[-110.73446875,105.130765625,23],[0.0799073218916662,-0.093747683476307,0.755254017896815,-0.64375271665574],[0,0,0,0],[8.999999E+09,8.999999E+09,8.999999E+09,8.999999E+09,8.999999E+09,8.999999E+09]];
	LOCAL CONST Robtarget Tr_meulage_bavure_P160 :=[[-108.04696875,105.8845859375,23],[0.0782084055442375,-0.0921215514798646,0.756740191543273,-0.642449490277812],[0,0,0,0],[8.999999E+09,8.999999E+09,8.999999E+09,8.999999E+09,8.999999E+09,8.999999E+09]];
	LOCAL CONST Robtarget Tr_meulage_bavure_P161 :=[[-107.098203125,106.097140625,23],[0.0772586675587503,-0.0913673505464314,0.758115325701143,-0.641049341687691],[0,0,0,0],[8.999999E+09,8.999999E+09,8.999999E+09,8.999999E+09,8.999999E+09,8.999999E+09]];
	LOCAL CONST Robtarget Tr_meulage_bavure_P162 :=[[-106.1117890625,106.3694765625,23],[0.0771689890904956,-0.0916163562192646,0.759328629402659,-0.639586915880348],[0,0,0,0],[8.999999E+09,8.999999E+09,8.999999E+09,8.999999E+09,8.999999E+09,8.999999E+09]];
	LOCAL CONST Robtarget Tr_meulage_bavure_P163 :=[[-102.4179375,107.152984375,23],[0.0777975054213532,-0.0926974815527003,0.760353365178672,-0.638135945645965],[0,0,0,0],[8.999999E+09,8.999999E+09,8.999999E+09,8.999999E+09,8.999999E+09,8.999999E+09]];
	LOCAL CONST Robtarget Tr_meulage_bavure_P164 :=[[-96.001796875,108.7913203125,23],[0.0787517821444272,-0.0941424622426149,0.761219570295702,-0.636773208772795],[0,0,0,0],[8.999999E+09,8.999999E+09,8.999999E+09,8.999999E+09,8.999999E+09,8.999999E+09]];
	LOCAL CONST Robtarget Tr_meulage_bavure_P165 :=[[-95.6863125,108.857328125,23],[0.0795259752587769,-0.0953345897819135,0.761961512284009,-0.635611193299898],[0,0,0,0],[8.999999E+09,8.999999E+09,8.999999E+09,8.999999E+09,8.999999E+09,8.999999E+09]];
	LOCAL CONST Robtarget Tr_meulage_bavure_P166 :=[[-95.5544140625,108.8944375,23],[0.0796591093804278,-0.0957070353485965,0.762621243423289,-0.634746743793945],[0,0,0,0],[8.999999E+09,8.999999E+09,8.999999E+09,8.999999E+09,8.999999E+09,8.999999E+09]];
	LOCAL CONST Robtarget Tr_meulage_bavure_P167 :=[[-95.090421875,109.0003671875,23],[0.0788841371264141,-0.094924708515954,0.763215879317989,-0.634246099065537],[0,0,0,0],[8.999999E+09,8.999999E+09,8.999999E+09,8.999999E+09,8.999999E+09,8.999999E+09]];
	LOCAL CONST Robtarget Tr_meulage_bavure_P168 :=[[-91.5986328125,109.6902734375,23],[0.0771899264376059,-0.0929645855860845,0.763724705880648,-0.634132379484664],[0,0,0,0],[8.999999E+09,8.999999E+09,8.999999E+09,8.999999E+09,8.999999E+09,8.999999E+09]];
	LOCAL CONST Robtarget Tr_meulage_bavure_P169 :=[[-88.8564140625,110.2953828125,23],[0.0747627327751832,-0.0900543093446174,0.764118771450325,-0.634368393186244],[0,0,0,0],[8.999999E+09,8.999999E+09,8.999999E+09,8.999999E+09,8.999999E+09,8.999999E+09]];
	LOCAL CONST Robtarget Tr_meulage_bavure_P170 :=[[-87.1766953125,110.5744609375,23],[0.0718868358836466,-0.0865343491517663,0.764321533022971,-0.634946205123657],[0,0,0,0],[8.999999E+09,8.999999E+09,8.999999E+09,8.999999E+09,8.999999E+09,8.999999E+09]];
	LOCAL CONST Robtarget Tr_meulage_bavure_P171 :=[[-86.382875,110.6813984375,23],[0.0687836500890445,-0.082684560325113,0.764310921822963,-0.635815136455875],[0,0,0,0],[8.999999E+09,8.999999E+09,8.999999E+09,8.999999E+09,8.999999E+09,8.999999E+09]];
	LOCAL CONST Robtarget Tr_meulage_bavure_P172 :=[[-84.3604140625,111.1460234375,23],[0.0655283309572558,-0.0786111524409777,0.764096628180546,-0.636932231369223],[0,0,0,0],[8.999999E+09,8.999999E+09,8.999999E+09,8.999999E+09,8.999999E+09,8.999999E+09]];
	LOCAL CONST Robtarget Tr_meulage_bavure_P173 :=[[-81.9507421875,111.54440625,23],[0.0620931332223892,-0.074290503372455,0.763678939353464,-0.63829447867208],[0,0,0,0],[8.999999E+09,8.999999E+09,8.999999E+09,8.999999E+09,8.999999E+09,8.999999E+09]];
	LOCAL CONST Robtarget Tr_meulage_bavure_P174 :=[[-80.2645859375,111.9013359375,23],[0.0584368425983391,-0.0696892297205684,0.763081913636481,-0.639870721137463],[0,0,0,0],[8.999999E+09,8.999999E+09,8.999999E+09,8.999999E+09,8.999999E+09,8.999999E+09]];
	LOCAL CONST Robtarget Tr_meulage_bavure_P175 :=[[-76.942046875,112.4490625,23],[0.0546288193728383,-0.0649074959362028,0.762327878623339,-0.641606510673685],[0,0,0,0],[8.999999E+09,8.999999E+09,8.999999E+09,8.999999E+09,8.999999E+09,8.999999E+09]];
	LOCAL CONST Robtarget Tr_meulage_bavure_P176 :=[[-72.0895390625,113.4118984375,23],[0.050898058837029,-0.0602283282233736,0.761410333907275,-0.643456478330316],[0,0,0,0],[8.999999E+09,8.999999E+09,8.999999E+09,8.999999E+09,8.999999E+09,8.999999E+09]];
	LOCAL CONST Robtarget Tr_meulage_bavure_P177 :=[[-66.0881953125,114.3616953125,23],[0.0475863095349679,-0.0560664361222813,0.760345608754694,-0.645342275953499],[0,0,0,0],[8.999999E+09,8.999999E+09,8.999999E+09,8.999999E+09,8.999999E+09,8.999999E+09]];
	LOCAL CONST Robtarget Tr_meulage_bavure_P178 :=[[-63.444671875,114.719515625,23],[0.0450257960605396,-0.052809549833417,0.759124796365831,-0.647235175711304],[0,0,0,0],[8.999999E+09,8.999999E+09,8.999999E+09,8.999999E+09,8.999999E+09,8.999999E+09]];
